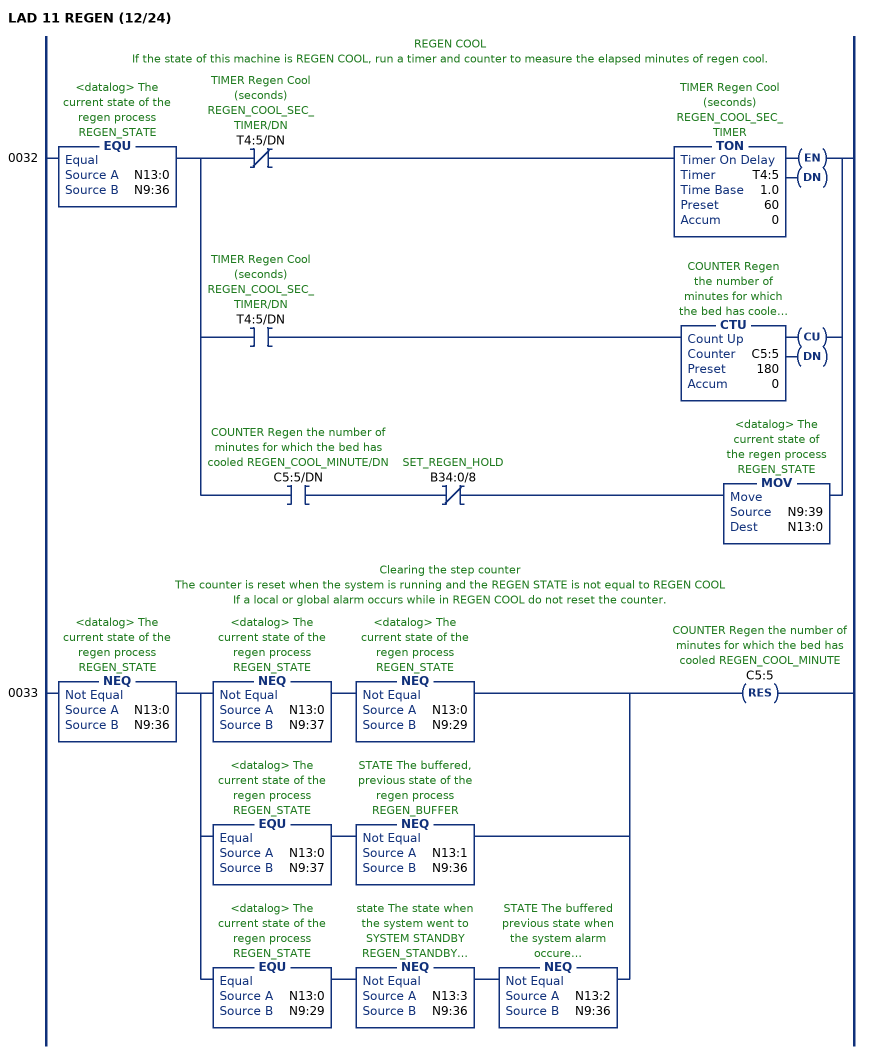
% Rung: 32 %
% REGEN COOL
% If the state of this machine is REGEN COOL, run a timer and counter to measure the elapsed minutes of regen cool. %
SOR EQU N13:0 N9:36 BST XIO T4:5/DN TON T4:5 1.0 60 0 NXB XIC T4:5/DN CTU C5:5 180 0 NXB XIC C5:5/DN XIO B34:0/8 MOV N9:39 N13:0 BND EOR
%   N13:0  REGEN_STATE  "<datalog> The current state of the regen process" %
%   N9:36  REGEN_COOL  "STATE Regen Cool" %
%   T4:5  REGEN_COOL_SEC_TIMER  "TIMER Regen Cool (seconds)" %
%   C5:5  REGEN_COOL_MINUTE  "COUNTER Regen the number of minutes for which the bed has cooled" %
%   B34:0/8  SET_REGEN_HOLD %
%   N9:39  REGEN_EQUALIZE %
% Rung: 33 %
% Clearing the step counter
% The counter is reset when the system is running and the REGEN STATE is not equal to REGEN COOL
% If a local or global alarm occurs while in REGEN COOL do not reset the counter. %
SOR NEQ N13:0 N9:36 BST NEQ N13:0 N9:37 NEQ N13:0 N9:29 NXB EQU N13:0 N9:37 NEQ N13:1 N9:36 NXB EQU N13:0 N9:29 NEQ N13:3 N9:36 NEQ N13:2 N9:36 BND RES C5:5 EOR
%   N13:0  REGEN_STATE  "<datalog> The current state of the regen process" %
%   N9:36  REGEN_COOL  "STATE Regen Cool" %
%   N9:37  REGEN_ALARM  "STATE Regen Alarm" %
%   N9:29  REGEN_IDLE %
%   N13:1  REGEN_BUFFER  "STATE The buffered, previous state of the regen process" %
%   N13:3  REGEN_STANDBY_BUFFER  "state The state when the system went to SYSTEM STANDBY" %
%   N13:2  REGEN_ALARM_BUFFER  "STATE The buffered previous state when the system alarm occured" %
%   C5:5  REGEN_COOL_MINUTE  "COUNTER Regen the number of minutes for which the bed has cooled" %

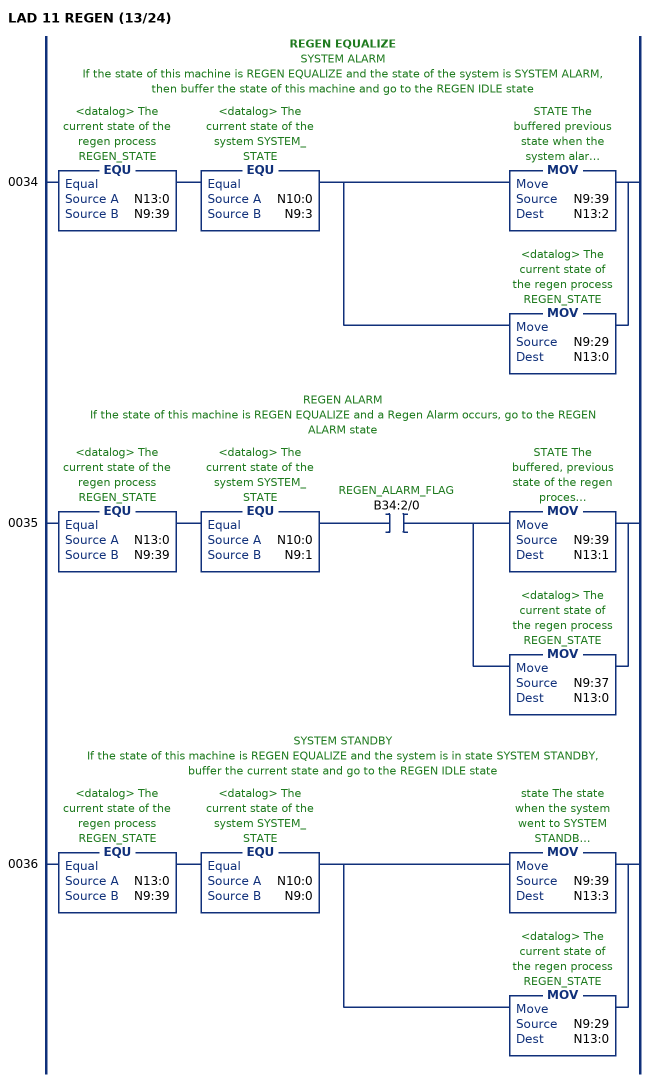
% Rung: 34 %
% TITLE: REGEN EQUALIZE %
% SYSTEM ALARM
% If the state of this machine is REGEN EQUALIZE and the state of the system is SYSTEM ALARM, then buffer the state of this machine and go to the REGEN IDLE state %
SOR EQU N13:0 N9:39 EQU N10:0 N9:3 BST MOV N9:39 N13:2 NXB MOV N9:29 N13:0 BND EOR
%   N13:0  REGEN_STATE  "<datalog> The current state of the regen process" %
%   N9:39  REGEN_EQUALIZE %
%   N10:0  SYSTEM_STATE  "<datalog> The current state of the system" %
%   N9:3  SYSTEM_ALARM  "STATE System Alarm" %
%   N13:2  REGEN_ALARM_BUFFER  "STATE The buffered previous state when the system alarm occured" %
%   N9:29  REGEN_IDLE %
% Rung: 35 %
% REGEN ALARM
% If the state of this machine is REGEN EQUALIZE and a Regen Alarm occurs, go to the REGEN ALARM state %
SOR EQU N13:0 N9:39 EQU N10:0 N9:1 XIC B34:2/0 BST MOV N9:39 N13:1 NXB MOV N9:37 N13:0 BND EOR
%   N13:0  REGEN_STATE  "<datalog> The current state of the regen process" %
%   N9:39  REGEN_EQUALIZE %
%   N10:0  SYSTEM_STATE  "<datalog> The current state of the system" %
%   N9:1  SYSTEM_PROCESS  "STATE System Process" %
%   B34:2/0  REGEN_ALARM_FLAG %
%   N13:1  REGEN_BUFFER  "STATE The buffered, previous state of the regen process" %
%   N9:37  REGEN_ALARM  "STATE Regen Alarm" %
% Rung: 36 %
% SYSTEM STANDBY
% If the state of this machine is REGEN EQUALIZE and the system is in state SYSTEM STANDBY, buffer the current state and go to the REGEN IDLE state %
SOR EQU N13:0 N9:39 EQU N10:0 N9:0 BST MOV N9:39 N13:3 NXB MOV N9:29 N13:0 BND EOR
%   N13:0  REGEN_STATE  "<datalog> The current state of the regen process" %
%   N9:39  REGEN_EQUALIZE %
%   N10:0  SYSTEM_STATE  "<datalog> The current state of the system" %
%   N9:0  SYSTEM_STANDBY  "STATE System Standby" %
%   N13:3  REGEN_STANDBY_BUFFER  "state The state when the system went to SYSTEM STANDBY" %
%   N9:29  REGEN_IDLE %

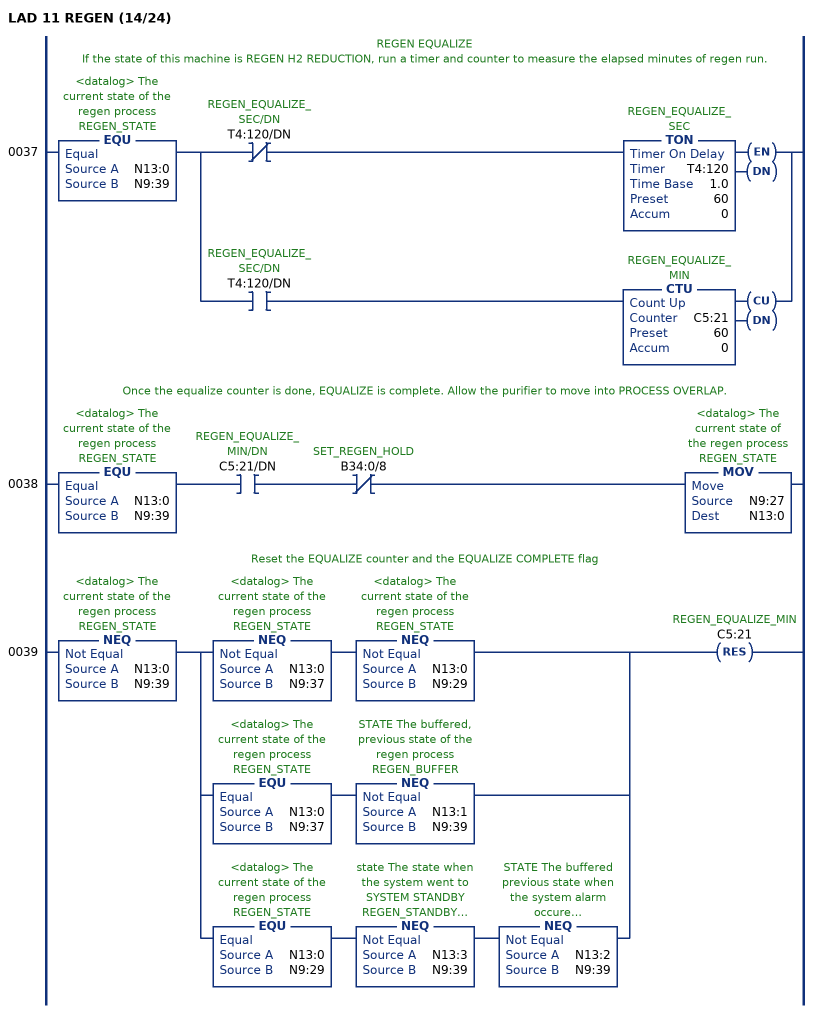
% Rung: 37 %
% REGEN EQUALIZE
% If the state of this machine is REGEN H2 REDUCTION, run a timer and counter to measure the elapsed minutes of regen run. %
SOR EQU N13:0 N9:39 BST XIO T4:120/DN TON T4:120 1.0 60 0 NXB XIC T4:120/DN CTU C5:21 60 0 BND EOR
%   N13:0  REGEN_STATE  "<datalog> The current state of the regen process" %
%   N9:39  REGEN_EQUALIZE %
%   T4:120  REGEN_EQUALIZE_SEC %
%   C5:21  REGEN_EQUALIZE_MIN %
% Rung: 38 %
% Once the equalize counter is done, EQUALIZE is complete. Allow the purifier to move into PROCESS OVERLAP. %
SOR EQU N13:0 N9:39 XIC C5:21/DN XIO B34:0/8 MOV N9:27 N13:0 EOR
%   N13:0  REGEN_STATE  "<datalog> The current state of the regen process" %
%   N9:39  REGEN_EQUALIZE %
%   C5:21  REGEN_EQUALIZE_MIN %
%   B34:0/8  SET_REGEN_HOLD %
%   N9:27  REGEN_CONDITION  "STATE Regen Idle" %
% Rung: 39 %
% Reset the EQUALIZE counter and the EQUALIZE COMPLETE flag %
SOR NEQ N13:0 N9:39 BST NEQ N13:0 N9:37 NEQ N13:0 N9:29 NXB EQU N13:0 N9:37 NEQ N13:1 N9:39 NXB EQU N13:0 N9:29 NEQ N13:3 N9:39 NEQ N13:2 N9:39 BND RES C5:21 EOR
%   N13:0  REGEN_STATE  "<datalog> The current state of the regen process" %
%   N9:39  REGEN_EQUALIZE %
%   N9:37  REGEN_ALARM  "STATE Regen Alarm" %
%   N9:29  REGEN_IDLE %
%   N13:1  REGEN_BUFFER  "STATE The buffered, previous state of the regen process" %
%   N13:3  REGEN_STANDBY_BUFFER  "state The state when the system went to SYSTEM STANDBY" %
%   N13:2  REGEN_ALARM_BUFFER  "STATE The buffered previous state when the system alarm occured" %
%   C5:21  REGEN_EQUALIZE_MIN %

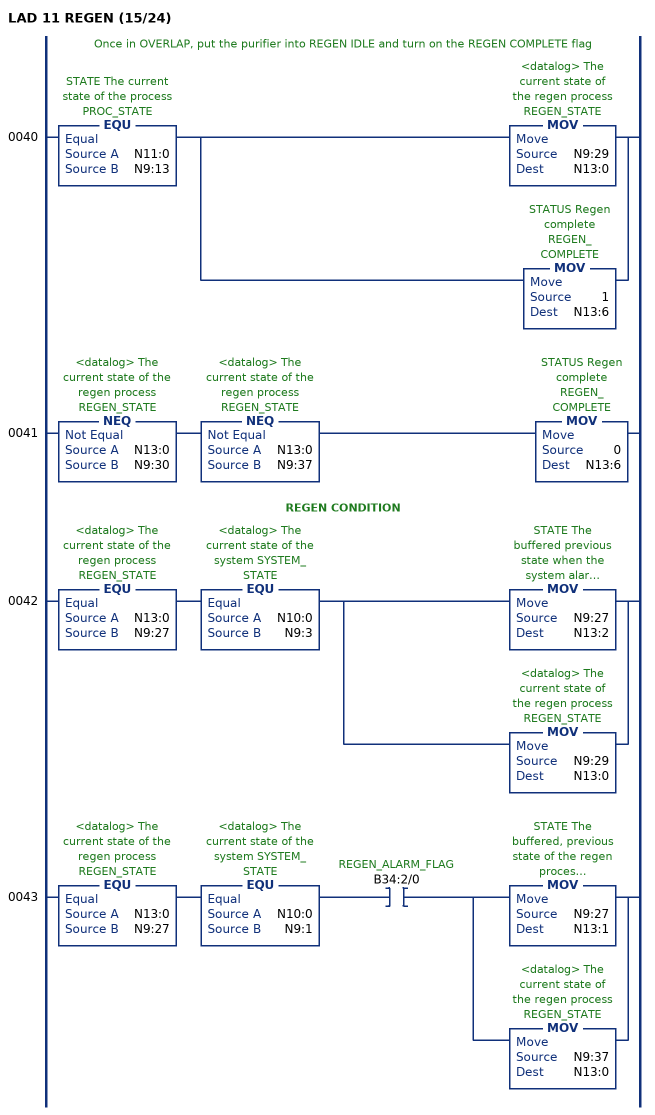
% Rung: 40 %
% Once in OVERLAP, put the purifier into REGEN IDLE and turn on the REGEN COMPLETE flag %
SOR EQU N11:0 N9:13 BST MOV N9:29 N13:0 NXB MOV 1 N13:6 BND EOR
%   N11:0  PROC_STATE  "STATE The current state of the process" %
%   N9:13  PROC_OVERLAP  "STATE Process Purify Overlap" %
%   N9:29  REGEN_IDLE %
%   N13:0  REGEN_STATE  "<datalog> The current state of the regen process" %
%   N13:6  REGEN_COMPLETE  "STATUS Regen complete" %
% Rung: 41 %
SOR NEQ N13:0 N9:30 NEQ N13:0 N9:37 MOV 0 N13:6 EOR
%   N13:0  REGEN_STATE  "<datalog> The current state of the regen process" %
%   N9:30  REGEN_STANDBY  "STATE Regen Standby" %
%   N9:37  REGEN_ALARM  "STATE Regen Alarm" %
%   N13:6  REGEN_COMPLETE  "STATUS Regen complete" %
% Rung: 42 %
% TITLE: REGEN CONDITION %
SOR EQU N13:0 N9:27 EQU N10:0 N9:3 BST MOV N9:27 N13:2 NXB MOV N9:29 N13:0 BND EOR
%   N13:0  REGEN_STATE  "<datalog> The current state of the regen process" %
%   N9:27  REGEN_CONDITION  "STATE Regen Idle" %
%   N10:0  SYSTEM_STATE  "<datalog> The current state of the system" %
%   N9:3  SYSTEM_ALARM  "STATE System Alarm" %
%   N13:2  REGEN_ALARM_BUFFER  "STATE The buffered previous state when the system alarm occured" %
%   N9:29  REGEN_IDLE %
% Rung: 43 %
SOR EQU N13:0 N9:27 EQU N10:0 N9:1 XIC B34:2/0 BST MOV N9:27 N13:1 NXB MOV N9:37 N13:0 BND EOR
%   N13:0  REGEN_STATE  "<datalog> The current state of the regen process" %
%   N9:27  REGEN_CONDITION  "STATE Regen Idle" %
%   N10:0  SYSTEM_STATE  "<datalog> The current state of the system" %
%   N9:1  SYSTEM_PROCESS  "STATE System Process" %
%   B34:2/0  REGEN_ALARM_FLAG %
%   N13:1  REGEN_BUFFER  "STATE The buffered, previous state of the regen process" %
%   N9:37  REGEN_ALARM  "STATE Regen Alarm" %

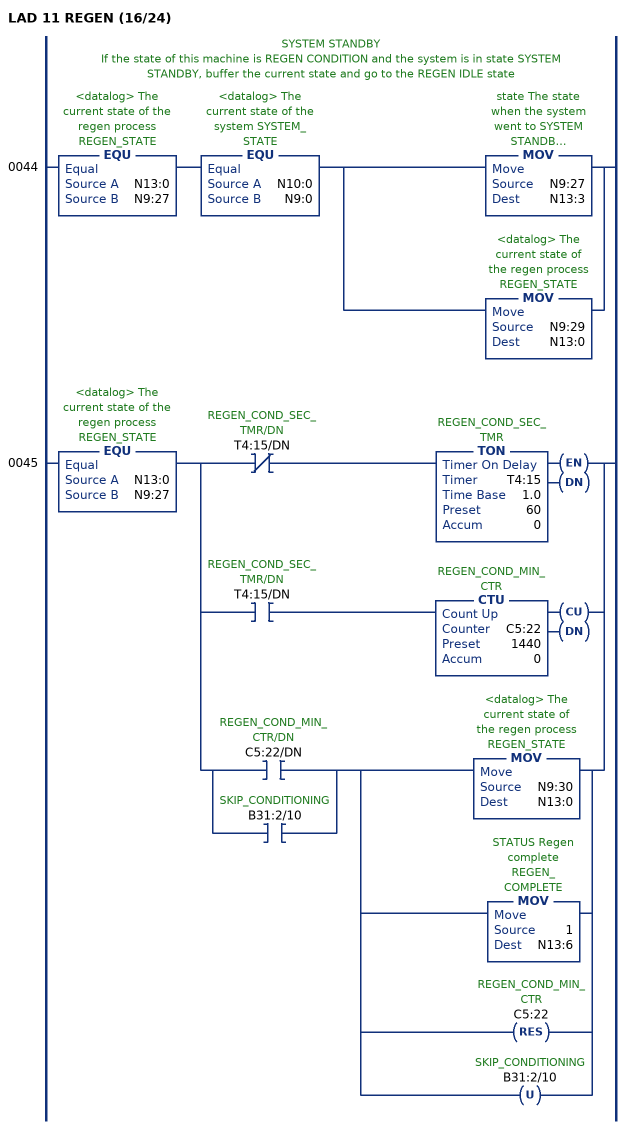
% Rung: 44 %
% SYSTEM STANDBY
% If the state of this machine is REGEN CONDITION and the system is in state SYSTEM STANDBY, buffer the current state and go to the REGEN IDLE state %
SOR EQU N13:0 N9:27 EQU N10:0 N9:0 BST MOV N9:27 N13:3 NXB MOV N9:29 N13:0 BND EOR
%   N13:0  REGEN_STATE  "<datalog> The current state of the regen process" %
%   N9:27  REGEN_CONDITION  "STATE Regen Idle" %
%   N10:0  SYSTEM_STATE  "<datalog> The current state of the system" %
%   N9:0  SYSTEM_STANDBY  "STATE System Standby" %
%   N13:3  REGEN_STANDBY_BUFFER  "state The state when the system went to SYSTEM STANDBY" %
%   N9:29  REGEN_IDLE %
% Rung: 45 %
SOR EQU N13:0 N9:27 BST XIO T4:15/DN TON T4:15 1.0 60 0 NXB XIC T4:15/DN CTU C5:22 1440 0 NXB BST XIC C5:22/DN NXB XIC B31:2/10 BND BST MOV N9:30 N13:0 NXB MOV 1 N13:6 NXB RES C5:22 NXB OTU B31:2/10 BND BND EOR
%   N13:0  REGEN_STATE  "<datalog> The current state of the regen process" %
%   N9:27  REGEN_CONDITION  "STATE Regen Idle" %
%   T4:15  REGEN_COND_SEC_TMR %
%   C5:22  REGEN_COND_MIN_CTR %
%   B31:2/10  SKIP_CONDITIONING %
%   N9:30  REGEN_STANDBY  "STATE Regen Standby" %
%   N13:6  REGEN_COMPLETE  "STATUS Regen complete" %

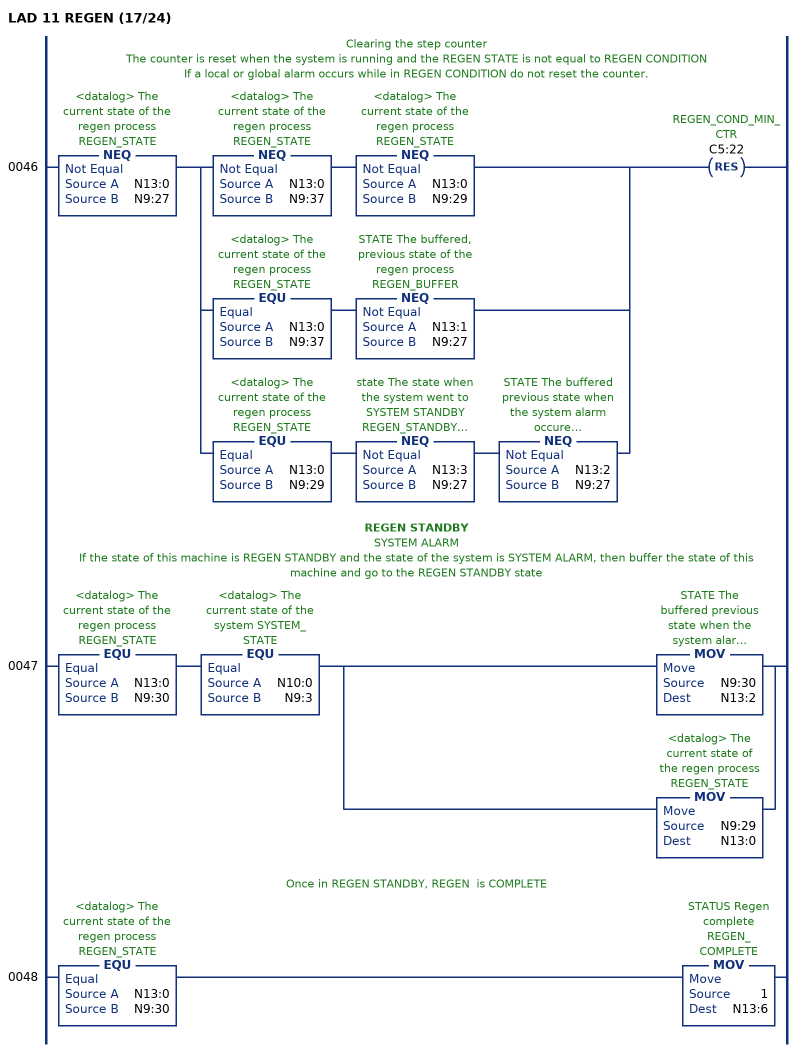
% Rung: 46 %
% Clearing the step counter
% The counter is reset when the system is running and the REGEN STATE is not equal to REGEN CONDITION
% If a local or global alarm occurs while in REGEN CONDITION do not reset the counter. %
SOR NEQ N13:0 N9:27 BST NEQ N13:0 N9:37 NEQ N13:0 N9:29 NXB EQU N13:0 N9:37 NEQ N13:1 N9:27 NXB EQU N13:0 N9:29 NEQ N13:3 N9:27 NEQ N13:2 N9:27 BND RES C5:22 EOR
%   N13:0  REGEN_STATE  "<datalog> The current state of the regen process" %
%   N9:27  REGEN_CONDITION  "STATE Regen Idle" %
%   N9:37  REGEN_ALARM  "STATE Regen Alarm" %
%   N9:29  REGEN_IDLE %
%   N13:1  REGEN_BUFFER  "STATE The buffered, previous state of the regen process" %
%   N13:3  REGEN_STANDBY_BUFFER  "state The state when the system went to SYSTEM STANDBY" %
%   N13:2  REGEN_ALARM_BUFFER  "STATE The buffered previous state when the system alarm occured" %
%   C5:22  REGEN_COND_MIN_CTR %
% Rung: 47 %
% TITLE: REGEN STANDBY %
% SYSTEM ALARM
% If the state of this machine is REGEN STANDBY and the state of the system is SYSTEM ALARM, then buffer the state of this machine and go to the REGEN STANDBY state %
SOR EQU N13:0 N9:30 EQU N10:0 N9:3 BST MOV N9:30 N13:2 NXB MOV N9:29 N13:0 BND EOR
%   N13:0  REGEN_STATE  "<datalog> The current state of the regen process" %
%   N9:30  REGEN_STANDBY  "STATE Regen Standby" %
%   N10:0  SYSTEM_STATE  "<datalog> The current state of the system" %
%   N9:3  SYSTEM_ALARM  "STATE System Alarm" %
%   N13:2  REGEN_ALARM_BUFFER  "STATE The buffered previous state when the system alarm occured" %
%   N9:29  REGEN_IDLE %
% Rung: 48 %
% Once in REGEN STANDBY, REGEN  is COMPLETE %
SOR EQU N13:0 N9:30 MOV 1 N13:6 EOR
%   N13:0  REGEN_STATE  "<datalog> The current state of the regen process" %
%   N9:30  REGEN_STANDBY  "STATE Regen Standby" %
%   N13:6  REGEN_COMPLETE  "STATUS Regen complete" %

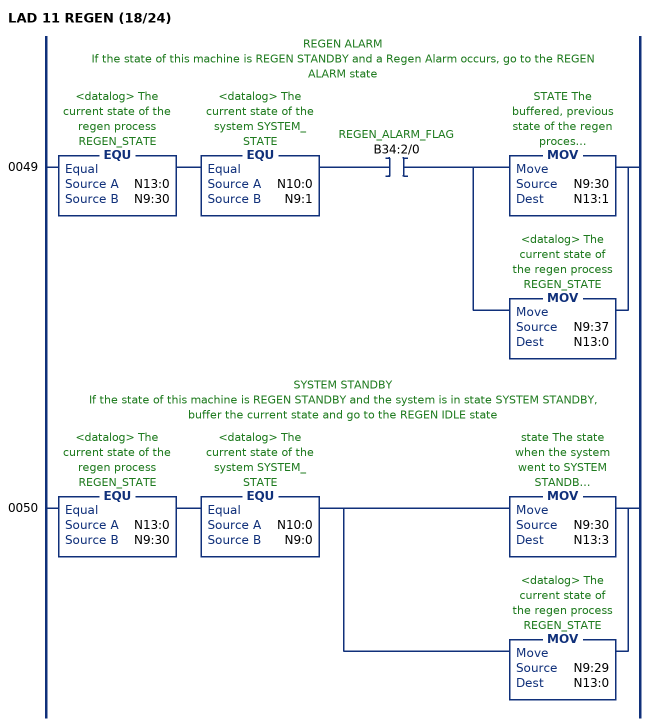
% Rung: 49 %
% REGEN ALARM
% If the state of this machine is REGEN STANDBY and a Regen Alarm occurs, go to the REGEN ALARM state %
SOR EQU N13:0 N9:30 EQU N10:0 N9:1 XIC B34:2/0 BST MOV N9:30 N13:1 NXB MOV N9:37 N13:0 BND EOR
%   N13:0  REGEN_STATE  "<datalog> The current state of the regen process" %
%   N9:30  REGEN_STANDBY  "STATE Regen Standby" %
%   N10:0  SYSTEM_STATE  "<datalog> The current state of the system" %
%   N9:1  SYSTEM_PROCESS  "STATE System Process" %
%   B34:2/0  REGEN_ALARM_FLAG %
%   N13:1  REGEN_BUFFER  "STATE The buffered, previous state of the regen process" %
%   N9:37  REGEN_ALARM  "STATE Regen Alarm" %
% Rung: 50 %
% SYSTEM STANDBY
% If the state of this machine is REGEN STANDBY and the system is in state SYSTEM STANDBY, buffer the current state and go to the REGEN IDLE state %
SOR EQU N13:0 N9:30 EQU N10:0 N9:0 BST MOV N9:30 N13:3 NXB MOV N9:29 N13:0 BND EOR
%   N13:0  REGEN_STATE  "<datalog> The current state of the regen process" %
%   N9:30  REGEN_STANDBY  "STATE Regen Standby" %
%   N10:0  SYSTEM_STATE  "<datalog> The current state of the system" %
%   N9:0  SYSTEM_STANDBY  "STATE System Standby" %
%   N13:3  REGEN_STANDBY_BUFFER  "state The state when the system went to SYSTEM STANDBY" %
%   N9:29  REGEN_IDLE %

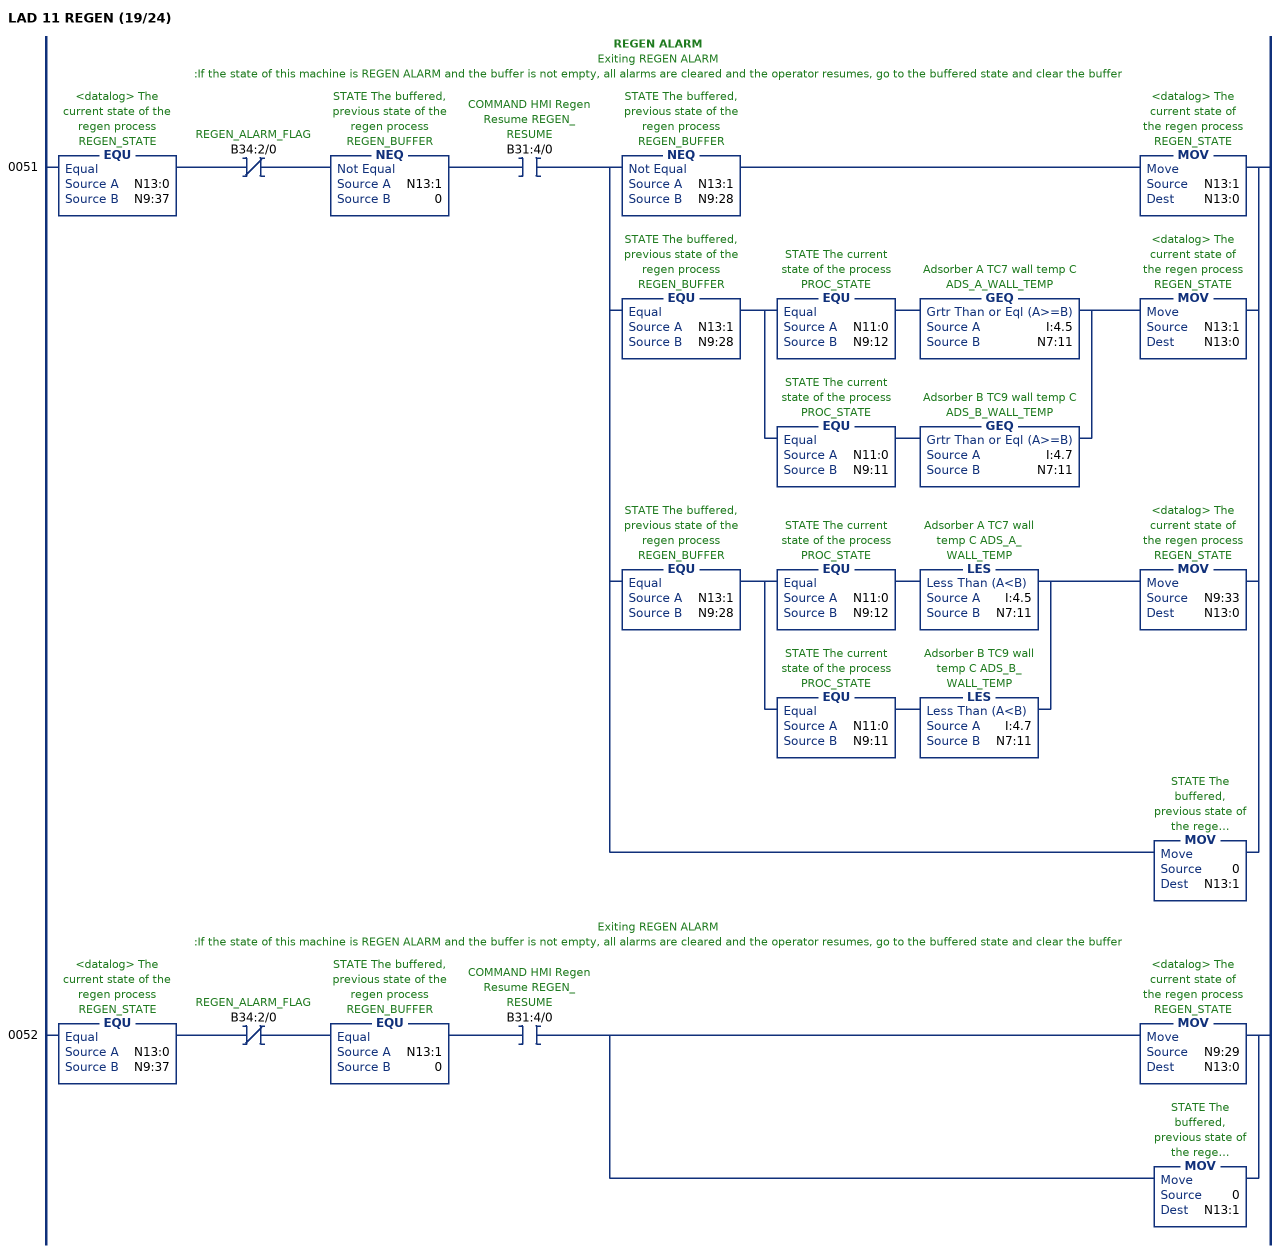
% Rung: 51 %
% TITLE: REGEN ALARM %
% Exiting REGEN ALARM
% :If the state of this machine is REGEN ALARM and the buffer is not empty, all alarms are cleared and the operator resumes, go to the buffered state and clear the buffer %
SOR EQU N13:0 N9:37 XIO B34:2/0 NEQ N13:1 0 XIC B31:4/0 BST NEQ N13:1 N9:28 MOV N13:1 N13:0 NXB EQU N13:1 N9:28 BST EQU N11:0 N9:12 GEQ I:4.5 N7:11 NXB EQU N11:0 N9:11 GEQ I:4.7 N7:11 BND MOV N13:1 N13:0 NXB EQU N13:1 N9:28 BST EQU N11:0 N9:12 LES I:4.5 N7:11 NXB EQU N11:0 N9:11 LES I:4.7 N7:11 BND MOV N9:33 N13:0 NXB MOV 0 N13:1 BND EOR
%   N13:0  REGEN_STATE  "<datalog> The current state of the regen process" %
%   N9:37  REGEN_ALARM  "STATE Regen Alarm" %
%   B34:2/0  REGEN_ALARM_FLAG %
%   N13:1  REGEN_BUFFER  "STATE The buffered, previous state of the regen process" %
%   B31:4/0  REGEN_RESUME  "COMMAND HMI Regen Resume" %
%   N9:28  REGEN_RUN %
%   N11:0  PROC_STATE  "STATE The current state of the process" %
%   N9:12  PROC_REGEN_A  "STATE Process Purify B" %
%   I:4.5  ADS_A_WALL_TEMP  "Adsorber A TC7 wall temp C" %
%   N7:11  ADS_BED_TEMP_HIGH  "CONFIG The temp at which the regen process may continue" %
%   N9:11  PROC_REGEN_B  "STATE Process Purify A" %
%   I:4.7  ADS_B_WALL_TEMP  "Adsorber B TC9 wall temp C" %
%   N9:33  REGEN_HEAT_BED  "STATE Regen Heat wall" %
% Rung: 52 %
% Exiting REGEN ALARM
% :If the state of this machine is REGEN ALARM and the buffer is not empty, all alarms are cleared and the operator resumes, go to the buffered state and clear the buffer %
SOR EQU N13:0 N9:37 XIO B34:2/0 EQU N13:1 0 XIC B31:4/0 BST MOV N9:29 N13:0 NXB MOV 0 N13:1 BND EOR
%   N13:0  REGEN_STATE  "<datalog> The current state of the regen process" %
%   N9:37  REGEN_ALARM  "STATE Regen Alarm" %
%   B34:2/0  REGEN_ALARM_FLAG %
%   N13:1  REGEN_BUFFER  "STATE The buffered, previous state of the regen process" %
%   B31:4/0  REGEN_RESUME  "COMMAND HMI Regen Resume" %
%   N9:29  REGEN_IDLE %

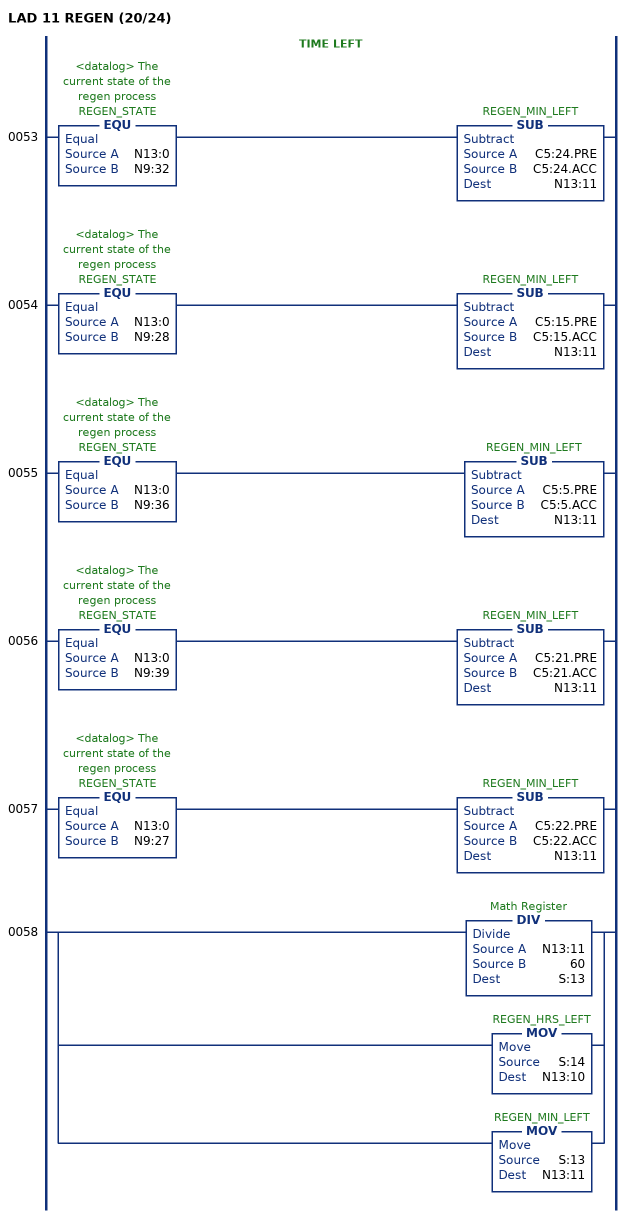
% Rung: 53 %
% TITLE: TIME LEFT %
SOR EQU N13:0 N9:32 SUB C5:24.PRE C5:24.ACC N13:11 EOR
%   N13:0  REGEN_STATE  "<datalog> The current state of the regen process" %
%   N9:32  REGEN_VENT  "STATE Regen Vent" %
%   C5:24  REGEN_VENT_MIN_CTR %
%   N13:11  REGEN_MIN_LEFT %
% Rung: 54 %
SOR EQU N13:0 N9:28 SUB C5:15.PRE C5:15.ACC N13:11 EOR
%   N13:0  REGEN_STATE  "<datalog> The current state of the regen process" %
%   N9:28  REGEN_RUN %
%   C5:15  REGEN_RUN_MINUTE %
%   N13:11  REGEN_MIN_LEFT %
% Rung: 55 %
SOR EQU N13:0 N9:36 SUB C5:5.PRE C5:5.ACC N13:11 EOR
%   N13:0  REGEN_STATE  "<datalog> The current state of the regen process" %
%   N9:36  REGEN_COOL  "STATE Regen Cool" %
%   C5:5  REGEN_COOL_MINUTE  "COUNTER Regen the number of minutes for which the bed has cooled" %
%   N13:11  REGEN_MIN_LEFT %
% Rung: 56 %
SOR EQU N13:0 N9:39 SUB C5:21.PRE C5:21.ACC N13:11 EOR
%   N13:0  REGEN_STATE  "<datalog> The current state of the regen process" %
%   N9:39  REGEN_EQUALIZE %
%   C5:21  REGEN_EQUALIZE_MIN %
%   N13:11  REGEN_MIN_LEFT %
% Rung: 57 %
SOR EQU N13:0 N9:27 SUB C5:22.PRE C5:22.ACC N13:11 EOR
%   N13:0  REGEN_STATE  "<datalog> The current state of the regen process" %
%   N9:27  REGEN_CONDITION  "STATE Regen Idle" %
%   C5:22  REGEN_COND_MIN_CTR %
%   N13:11  REGEN_MIN_LEFT %
% Rung: 58 %
SOR BST DIV N13:11 60 S:13 NXB MOV S:14 N13:10 NXB MOV S:13 N13:11 BND EOR
%   N13:11  REGEN_MIN_LEFT %
%   S:13  "Math Register" %
%   S:14  "Math Register" %
%   N13:10  REGEN_HRS_LEFT %

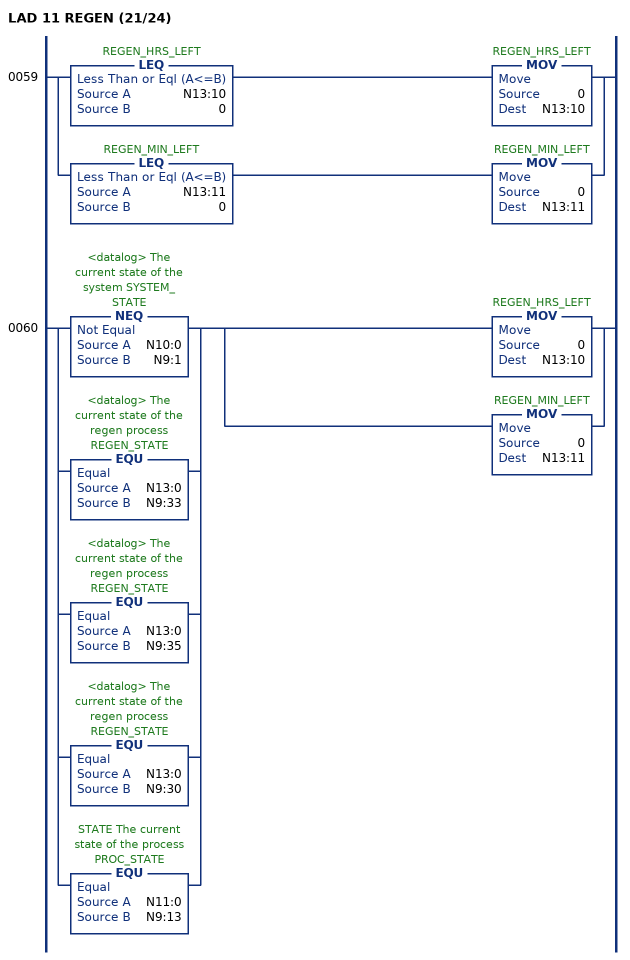
% Rung: 59 %
SOR BST LEQ N13:10 0 MOV 0 N13:10 NXB LEQ N13:11 0 MOV 0 N13:11 BND EOR
%   N13:10  REGEN_HRS_LEFT %
%   N13:11  REGEN_MIN_LEFT %
% Rung: 60 %
SOR BST NEQ N10:0 N9:1 NXB EQU N13:0 N9:33 NXB EQU N13:0 N9:35 NXB EQU N13:0 N9:30 NXB EQU N11:0 N9:13 BND BST MOV 0 N13:10 NXB MOV 0 N13:11 BND EOR
%   N10:0  SYSTEM_STATE  "<datalog> The current state of the system" %
%   N9:1  SYSTEM_PROCESS  "STATE System Process" %
%   N13:0  REGEN_STATE  "<datalog> The current state of the regen process" %
%   N9:33  REGEN_HEAT_BED  "STATE Regen Heat wall" %
%   N9:35  REGEN_COOL_WALL  "STATE Regen Cool wall" %
%   N9:30  REGEN_STANDBY  "STATE Regen Standby" %
%   N11:0  PROC_STATE  "STATE The current state of the process" %
%   N9:13  PROC_OVERLAP  "STATE Process Purify Overlap" %
%   N13:10  REGEN_HRS_LEFT %
%   N13:11  REGEN_MIN_LEFT %

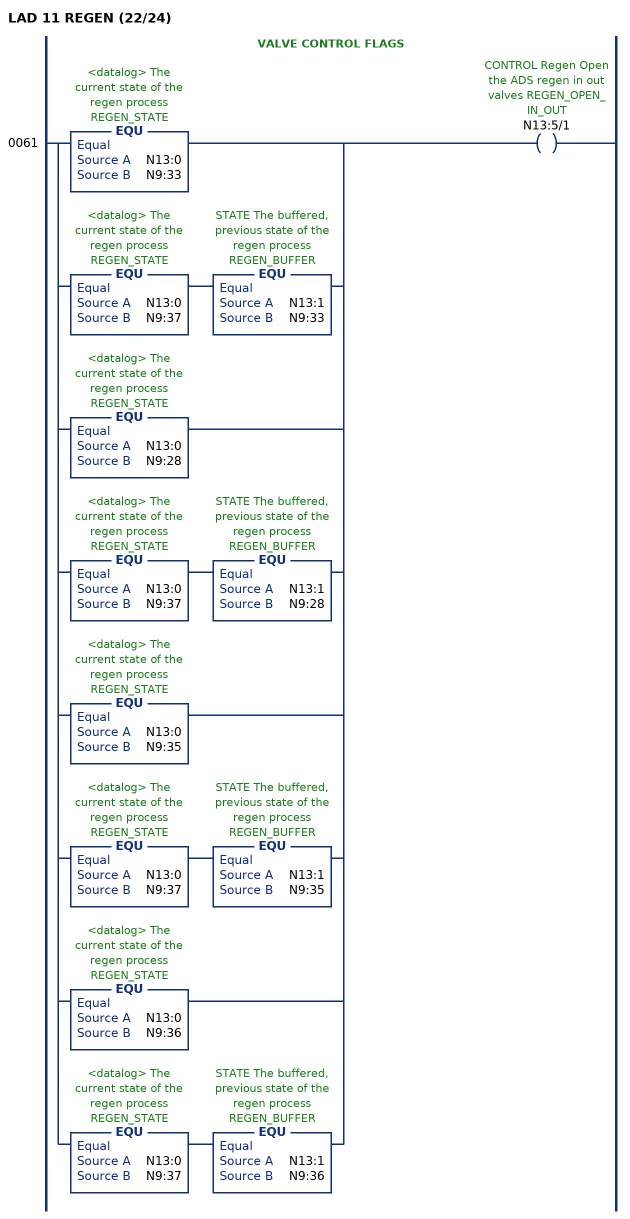
% Rung: 61 %
% TITLE: VALVE CONTROL FLAGS %
SOR BST EQU N13:0 N9:33 NXB EQU N13:0 N9:37 EQU N13:1 N9:33 NXB EQU N13:0 N9:28 NXB EQU N13:0 N9:37 EQU N13:1 N9:28 NXB EQU N13:0 N9:35 NXB EQU N13:0 N9:37 EQU N13:1 N9:35 NXB EQU N13:0 N9:36 NXB EQU N13:0 N9:37 EQU N13:1 N9:36 BND OTE N13:5/1 EOR
%   N13:0  REGEN_STATE  "<datalog> The current state of the regen process" %
%   N9:33  REGEN_HEAT_BED  "STATE Regen Heat wall" %
%   N9:37  REGEN_ALARM  "STATE Regen Alarm" %
%   N13:1  REGEN_BUFFER  "STATE The buffered, previous state of the regen process" %
%   N9:28  REGEN_RUN %
%   N9:35  REGEN_COOL_WALL  "STATE Regen Cool wall" %
%   N9:36  REGEN_COOL  "STATE Regen Cool" %
%   N13:5/1  REGEN_OPEN_IN_OUT  "CONTROL Regen Open the ADS regen in out valves" %

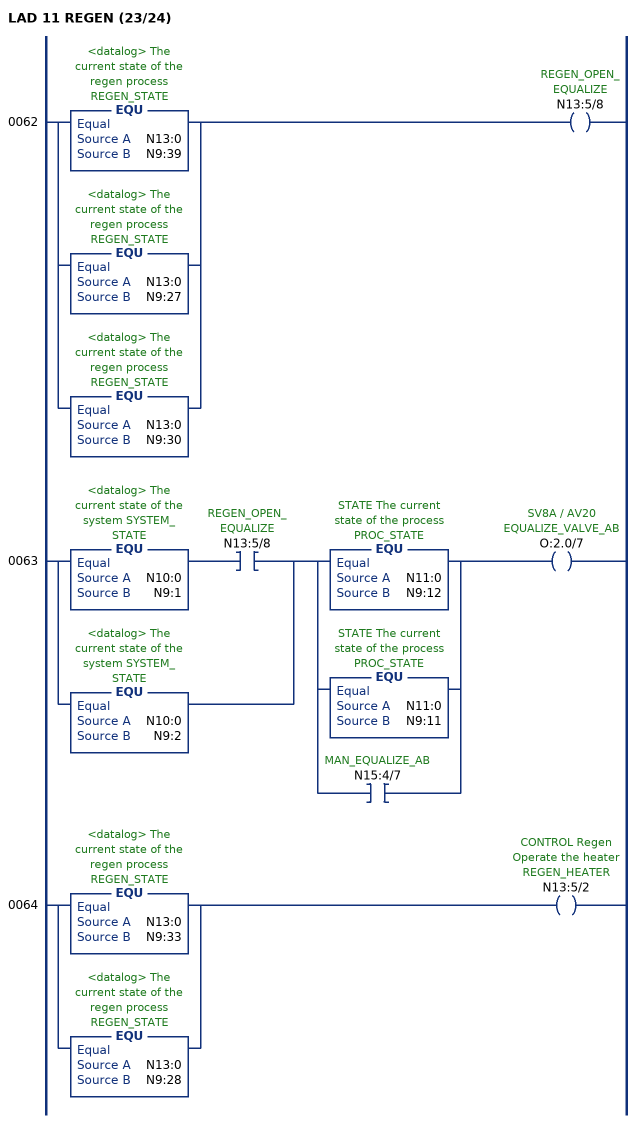
% Rung: 62 %
SOR BST EQU N13:0 N9:39 NXB EQU N13:0 N9:27 NXB EQU N13:0 N9:30 BND OTE N13:5/8 EOR
%   N13:0  REGEN_STATE  "<datalog> The current state of the regen process" %
%   N9:39  REGEN_EQUALIZE %
%   N9:27  REGEN_CONDITION  "STATE Regen Idle" %
%   N9:30  REGEN_STANDBY  "STATE Regen Standby" %
%   N13:5/8  REGEN_OPEN_EQUALIZE %
% Rung: 63 %
SOR BST EQU N10:0 N9:1 XIC N13:5/8 NXB EQU N10:0 N9:2 BND BST EQU N11:0 N9:12 NXB EQU N11:0 N9:11 NXB XIC N15:4/7 BND OTE O:2.0/7 EOR
%   N10:0  SYSTEM_STATE  "<datalog> The current state of the system" %
%   N9:1  SYSTEM_PROCESS  "STATE System Process" %
%   N13:5/8  REGEN_OPEN_EQUALIZE %
%   N9:2  SYSTEM_MANUAL  "STATE System Manual" %
%   N11:0  PROC_STATE  "STATE The current state of the process" %
%   N9:12  PROC_REGEN_A  "STATE Process Purify B" %
%   N9:11  PROC_REGEN_B  "STATE Process Purify A" %
%   N15:4/7  MAN_EQUALIZE_AB %
%   O:2.0/7  EQUALIZE_VALVE_AB  "SV8A / AV20" %
% Rung: 64 %
SOR BST EQU N13:0 N9:33 NXB EQU N13:0 N9:28 BND OTE N13:5/2 EOR
%   N13:0  REGEN_STATE  "<datalog> The current state of the regen process" %
%   N9:33  REGEN_HEAT_BED  "STATE Regen Heat wall" %
%   N9:28  REGEN_RUN %
%   N13:5/2  REGEN_HEATER  "CONTROL Regen Operate the heater" %

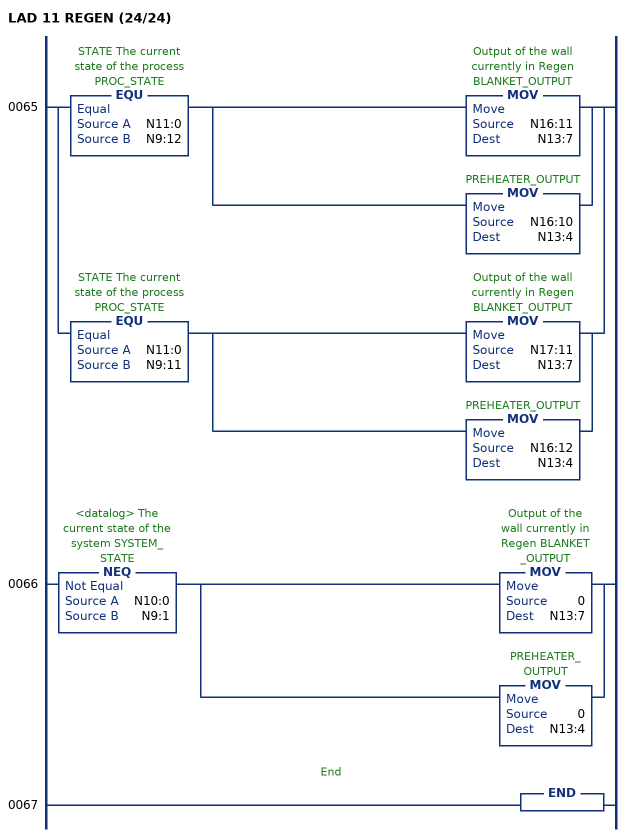
% Rung: 65 %
SOR BST EQU N11:0 N9:12 BST MOV N16:11 N13:7 NXB MOV N16:10 N13:4 BND NXB EQU N11:0 N9:11 BST MOV N17:11 N13:7 NXB MOV N16:12 N13:4 BND BND EOR
%   N11:0  PROC_STATE  "STATE The current state of the process" %
%   N9:12  PROC_REGEN_A  "STATE Process Purify B" %
%   N16:11  ADS_A_BLNKT_OUTPUT  "CONTROL ADS A Blanket output (percent)" %
%   N13:7  BLANKET_OUTPUT  "Output of the wall currently in Regen" %
%   N16:10  ADS_A_PH_OUTPUT  "<datalog> Adsorber A heater duty cycle %" %
%   N13:4  PREHEATER_OUTPUT %
%   N9:11  PROC_REGEN_B  "STATE Process Purify A" %
%   N17:11  ADS_B_BLNKT_OUTPUT  "CONTROL ADS A Blanket output" %
%   N16:12  ADS_B_PH_OUTPUT  "<datalog> Adsorber B heater duty cycle %" %
% Rung: 66 %
SOR NEQ N10:0 N9:1 BST MOV 0 N13:7 NXB MOV 0 N13:4 BND EOR
%   N10:0  SYSTEM_STATE  "<datalog> The current state of the system" %
%   N9:1  SYSTEM_PROCESS  "STATE System Process" %
%   N13:7  BLANKET_OUTPUT  "Output of the wall currently in Regen" %
%   N13:4  PREHEATER_OUTPUT %
% Rung: 67 %
% End %
SOR END EOR

LADDER 12 "REGEN_FLT"    % regen alarms and warnings %
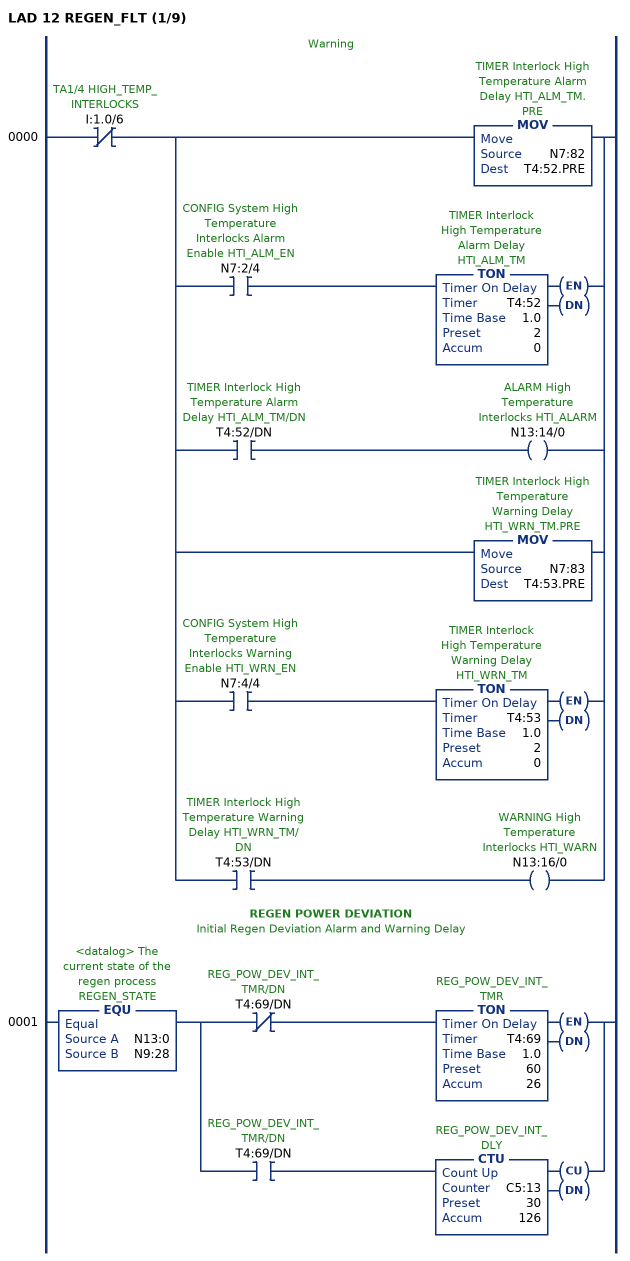
% Rung: 0 %
% Warning %
SOR XIO I:1.0/6 BST MOV N7:82 T4:52.PRE NXB XIC N7:2/4 TON T4:52 1.0 2 0 NXB XIC T4:52/DN OTE N13:14/0 NXB MOV N7:83 T4:53.PRE NXB XIC N7:4/4 TON T4:53 1.0 2 0 NXB XIC T4:53/DN OTE N13:16/0 BND EOR
%   I:1.0/6  HIGH_TEMP_INTERLOCKS  "TA1/4" %
%   N7:82  HTI_ALM_DY  "CONFIG Interlocks High Temp Alarm Delay" %
%   T4:52  HTI_ALM_TM  "TIMER Interlock High Temperature Alarm Delay" %
%   N7:2/4  HTI_ALM_EN  "CONFIG System High Temperature Interlocks Alarm Enable" %
%   N13:14/0  HTI_ALARM  "ALARM High Temperature Interlocks" %
%   N7:83  HTI_WRN_DY  "CONFIG Interlocks High Temp Warning Delay" %
%   T4:53  HTI_WRN_TM  "TIMER Interlock High Temperature Warning Delay" %
%   N7:4/4  HTI_WRN_EN  "CONFIG System High Temperature Interlocks Warning Enable" %
%   N13:16/0  HTI_WARN  "WARNING High Temperature Interlocks" %
% Rung: 1 %
% TITLE: REGEN POWER DEVIATION %
% Initial Regen Deviation Alarm and Warning Delay %
SOR EQU N13:0 N9:28 BST XIO T4:69/DN TON T4:69 1.0 60 26 NXB XIC T4:69/DN CTU C5:13 30 126 BND EOR
%   N13:0  REGEN_STATE  "<datalog> The current state of the regen process" %
%   N9:28  REGEN_RUN %
%   T4:69  REG_POW_DEV_INT_TMR %
%   C5:13  REG_POW_DEV_INT_DLY %

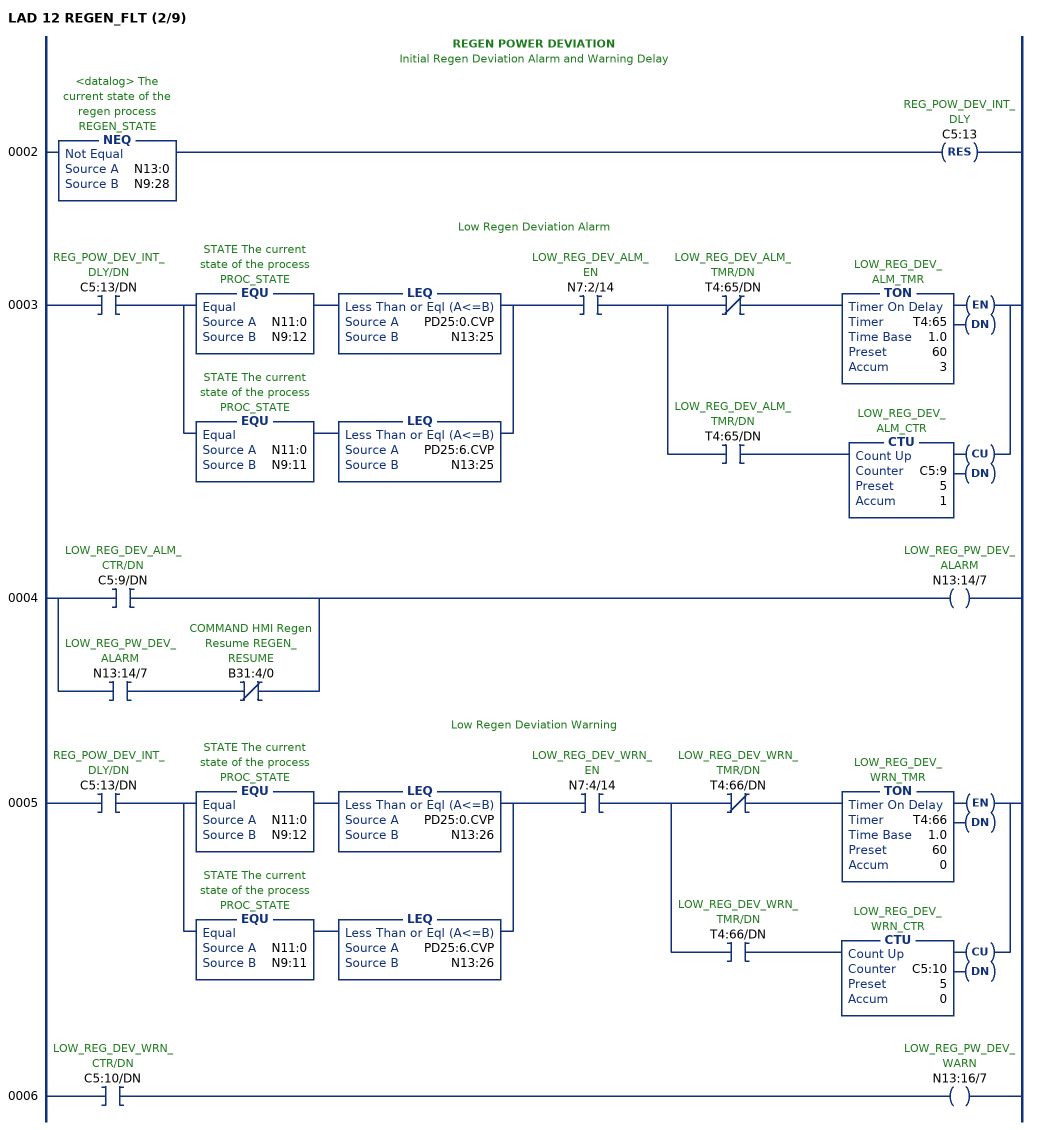
% Rung: 2 %
% TITLE: REGEN POWER DEVIATION %
% Initial Regen Deviation Alarm and Warning Delay %
SOR NEQ N13:0 N9:28 RES C5:13 EOR
%   N13:0  REGEN_STATE  "<datalog> The current state of the regen process" %
%   N9:28  REGEN_RUN %
%   C5:13  REG_POW_DEV_INT_DLY %
% Rung: 3 %
% Low Regen Deviation Alarm %
SOR XIC C5:13/DN BST EQU N11:0 N9:12 LEQ PD25:0.CVP N13:25 NXB EQU N11:0 N9:11 LEQ PD25:6.CVP N13:25 BND XIC N7:2/14 BST XIO T4:65/DN TON T4:65 1.0 60 3 NXB XIC T4:65/DN CTU C5:9 5 1 BND EOR
%   C5:13  REG_POW_DEV_INT_DLY %
%   N11:0  PROC_STATE  "STATE The current state of the process" %
%   N9:12  PROC_REGEN_A  "STATE Process Purify B" %
%   N13:25  LOW_REG_DEV_ALM_SP %
%   N9:11  PROC_REGEN_B  "STATE Process Purify A" %
%   N7:2/14  LOW_REG_DEV_ALM_EN %
%   T4:65  LOW_REG_DEV_ALM_TMR %
%   C5:9  LOW_REG_DEV_ALM_CTR %
% Rung: 4 %
SOR BST XIC C5:9/DN NXB XIC N13:14/7 XIO B31:4/0 BND OTE N13:14/7 EOR
%   C5:9  LOW_REG_DEV_ALM_CTR %
%   N13:14/7  LOW_REG_PW_DEV_ALARM %
%   B31:4/0  REGEN_RESUME  "COMMAND HMI Regen Resume" %
% Rung: 5 %
% Low Regen Deviation Warning %
SOR XIC C5:13/DN BST EQU N11:0 N9:12 LEQ PD25:0.CVP N13:26 NXB EQU N11:0 N9:11 LEQ PD25:6.CVP N13:26 BND XIC N7:4/14 BST XIO T4:66/DN TON T4:66 1.0 60 0 NXB XIC T4:66/DN CTU C5:10 5 0 BND EOR
%   C5:13  REG_POW_DEV_INT_DLY %
%   N11:0  PROC_STATE  "STATE The current state of the process" %
%   N9:12  PROC_REGEN_A  "STATE Process Purify B" %
%   N13:26  LOW_REG_DEV_WRN_SP %
%   N9:11  PROC_REGEN_B  "STATE Process Purify A" %
%   N7:4/14  LOW_REG_DEV_WRN_EN %
%   T4:66  LOW_REG_DEV_WRN_TMR %
%   C5:10  LOW_REG_DEV_WRN_CTR %
% Rung: 6 %
SOR XIC C5:10/DN OTE N13:16/7 EOR
%   C5:10  LOW_REG_DEV_WRN_CTR %
%   N13:16/7  LOW_REG_PW_DEV_WARN %

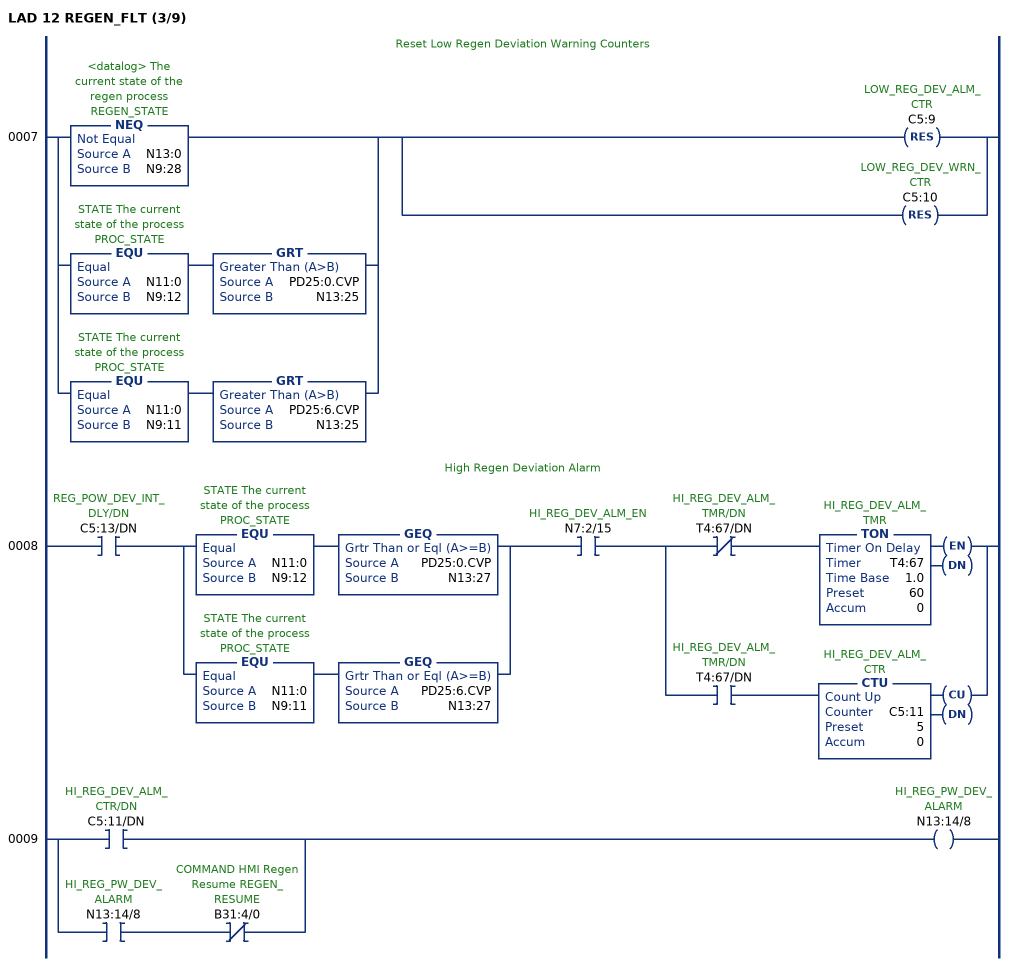
% Rung: 7 %
% Reset Low Regen Deviation Warning Counters %
SOR BST NEQ N13:0 N9:28 NXB EQU N11:0 N9:12 GRT PD25:0.CVP N13:25 NXB EQU N11:0 N9:11 GRT PD25:6.CVP N13:25 BND BST RES C5:9 NXB RES C5:10 BND EOR
%   N13:0  REGEN_STATE  "<datalog> The current state of the regen process" %
%   N9:28  REGEN_RUN %
%   N11:0  PROC_STATE  "STATE The current state of the process" %
%   N9:12  PROC_REGEN_A  "STATE Process Purify B" %
%   N13:25  LOW_REG_DEV_ALM_SP %
%   N9:11  PROC_REGEN_B  "STATE Process Purify A" %
%   C5:9  LOW_REG_DEV_ALM_CTR %
%   C5:10  LOW_REG_DEV_WRN_CTR %
% Rung: 8 %
% High Regen Deviation Alarm %
SOR XIC C5:13/DN BST EQU N11:0 N9:12 GEQ PD25:0.CVP N13:27 NXB EQU N11:0 N9:11 GEQ PD25:6.CVP N13:27 BND XIC N7:2/15 BST XIO T4:67/DN TON T4:67 1.0 60 0 NXB XIC T4:67/DN CTU C5:11 5 0 BND EOR
%   C5:13  REG_POW_DEV_INT_DLY %
%   N11:0  PROC_STATE  "STATE The current state of the process" %
%   N9:12  PROC_REGEN_A  "STATE Process Purify B" %
%   N13:27  HI_REG_DEV_ALM_SP %
%   N9:11  PROC_REGEN_B  "STATE Process Purify A" %
%   N7:2/15  HI_REG_DEV_ALM_EN %
%   T4:67  HI_REG_DEV_ALM_TMR %
%   C5:11  HI_REG_DEV_ALM_CTR %
% Rung: 9 %
SOR BST XIC C5:11/DN NXB XIC N13:14/8 XIO B31:4/0 BND OTE N13:14/8 EOR
%   C5:11  HI_REG_DEV_ALM_CTR %
%   N13:14/8  HI_REG_PW_DEV_ALARM %
%   B31:4/0  REGEN_RESUME  "COMMAND HMI Regen Resume" %

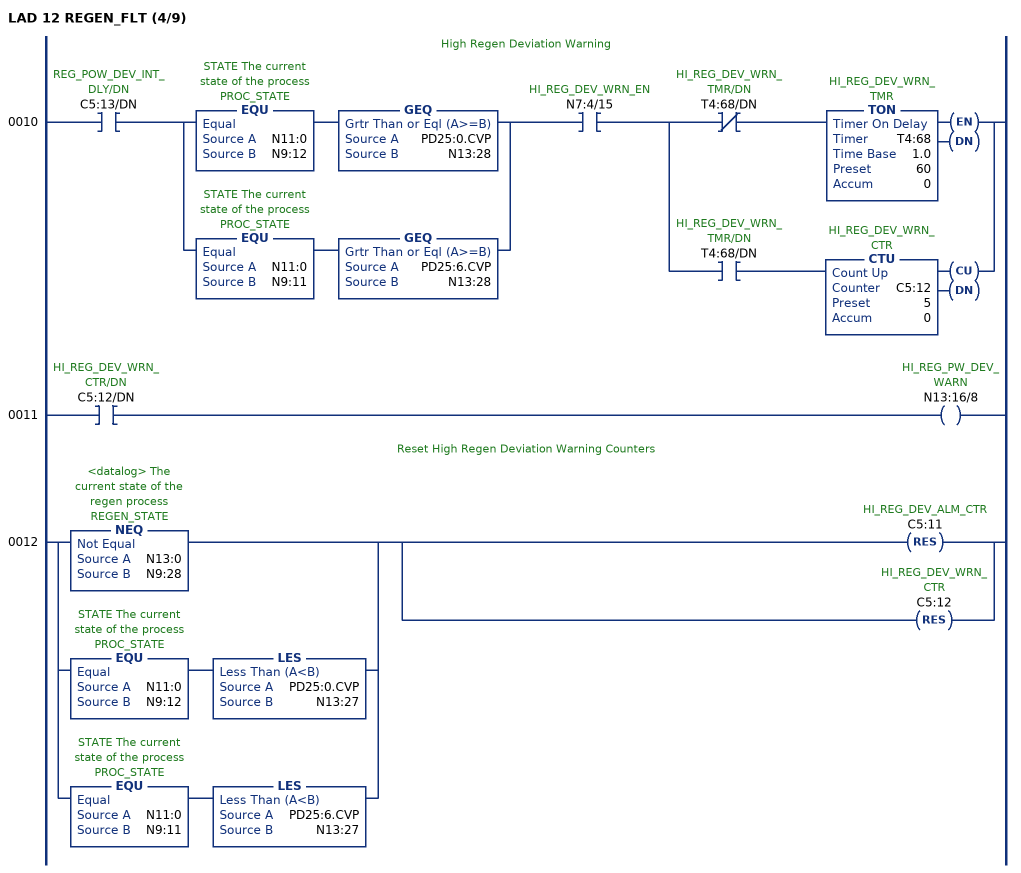
% Rung: 10 %
% High Regen Deviation Warning %
SOR XIC C5:13/DN BST EQU N11:0 N9:12 GEQ PD25:0.CVP N13:28 NXB EQU N11:0 N9:11 GEQ PD25:6.CVP N13:28 BND XIC N7:4/15 BST XIO T4:68/DN TON T4:68 1.0 60 0 NXB XIC T4:68/DN CTU C5:12 5 0 BND EOR
%   C5:13  REG_POW_DEV_INT_DLY %
%   N11:0  PROC_STATE  "STATE The current state of the process" %
%   N9:12  PROC_REGEN_A  "STATE Process Purify B" %
%   N13:28  HI_REG_DEV_WRN_SP %
%   N9:11  PROC_REGEN_B  "STATE Process Purify A" %
%   N7:4/15  HI_REG_DEV_WRN_EN %
%   T4:68  HI_REG_DEV_WRN_TMR %
%   C5:12  HI_REG_DEV_WRN_CTR %
% Rung: 11 %
SOR XIC C5:12/DN OTE N13:16/8 EOR
%   C5:12  HI_REG_DEV_WRN_CTR %
%   N13:16/8  HI_REG_PW_DEV_WARN %
% Rung: 12 %
% Reset High Regen Deviation Warning Counters %
SOR BST NEQ N13:0 N9:28 NXB EQU N11:0 N9:12 LES PD25:0.CVP N13:27 NXB EQU N11:0 N9:11 LES PD25:6.CVP N13:27 BND BST RES C5:11 NXB RES C5:12 BND EOR
%   N13:0  REGEN_STATE  "<datalog> The current state of the regen process" %
%   N9:28  REGEN_RUN %
%   N11:0  PROC_STATE  "STATE The current state of the process" %
%   N9:12  PROC_REGEN_A  "STATE Process Purify B" %
%   N13:27  HI_REG_DEV_ALM_SP %
%   N9:11  PROC_REGEN_B  "STATE Process Purify A" %
%   C5:11  HI_REG_DEV_ALM_CTR %
%   C5:12  HI_REG_DEV_WRN_CTR %

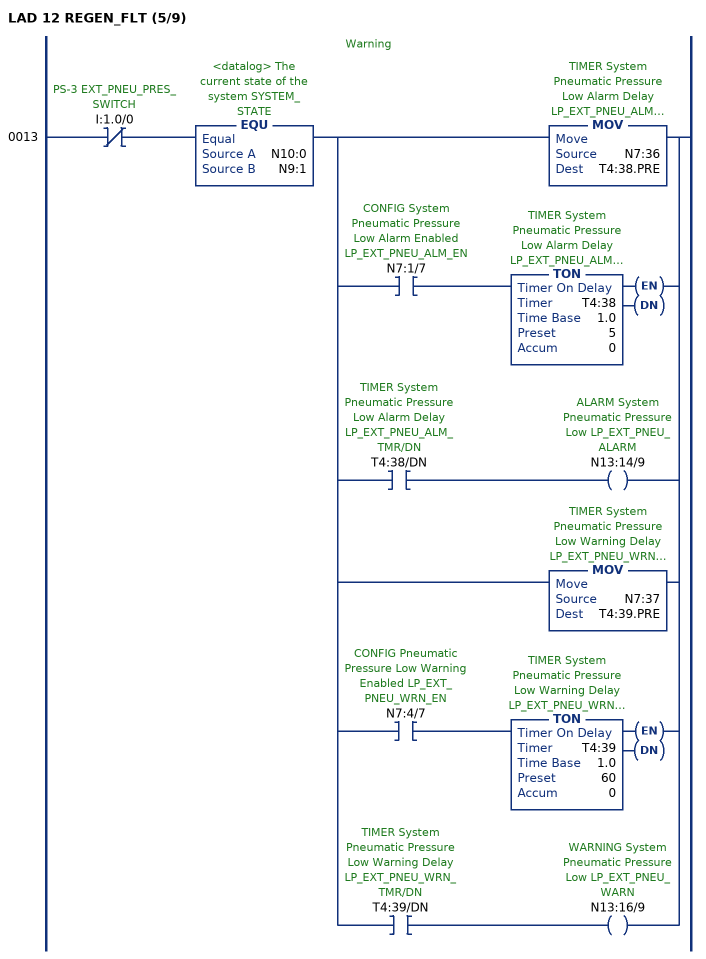
% Rung: 13 %
% Warning %
SOR XIO I:1.0/0 EQU N10:0 N9:1 BST MOV N7:36 T4:38.PRE NXB XIC N7:1/7 TON T4:38 1.0 5 0 NXB XIC T4:38/DN OTE N13:14/9 NXB MOV N7:37 T4:39.PRE NXB XIC N7:4/7 TON T4:39 1.0 60 0 NXB XIC T4:39/DN OTE N13:16/9 BND EOR
%   I:1.0/0  EXT_PNEU_PRES_SWITCH  "PS-3" %
%   N10:0  SYSTEM_STATE  "<datalog> The current state of the system" %
%   N9:1  SYSTEM_PROCESS  "STATE System Process" %
%   N7:36  LP_EXT_PNEU_ALM_DLY  "CONFIG Pneumatic Pressure Low Alarm Delay" %
%   T4:38  LP_EXT_PNEU_ALM_TMR  "TIMER System Pneumatic Pressure Low Alarm Delay" %
%   N7:1/7  LP_EXT_PNEU_ALM_EN  "CONFIG System Pneumatic Pressure Low Alarm Enabled" %
%   N13:14/9  LP_EXT_PNEU_ALARM  "ALARM System Pneumatic Pressure Low" %
%   N7:37  LP_EXT_PNEU_WRN_DLY  "CONFIG Pneumatic Pressure Low Warning Delay" %
%   T4:39  LP_EXT_PNEU_WRN_TMR  "TIMER System Pneumatic Pressure Low Warning Delay" %
%   N7:4/7  LP_EXT_PNEU_WRN_EN  "CONFIG Pneumatic Pressure Low Warning Enabled" %
%   N13:16/9  LP_EXT_PNEU_WARN  "WARNING System Pneumatic Pressure Low" %

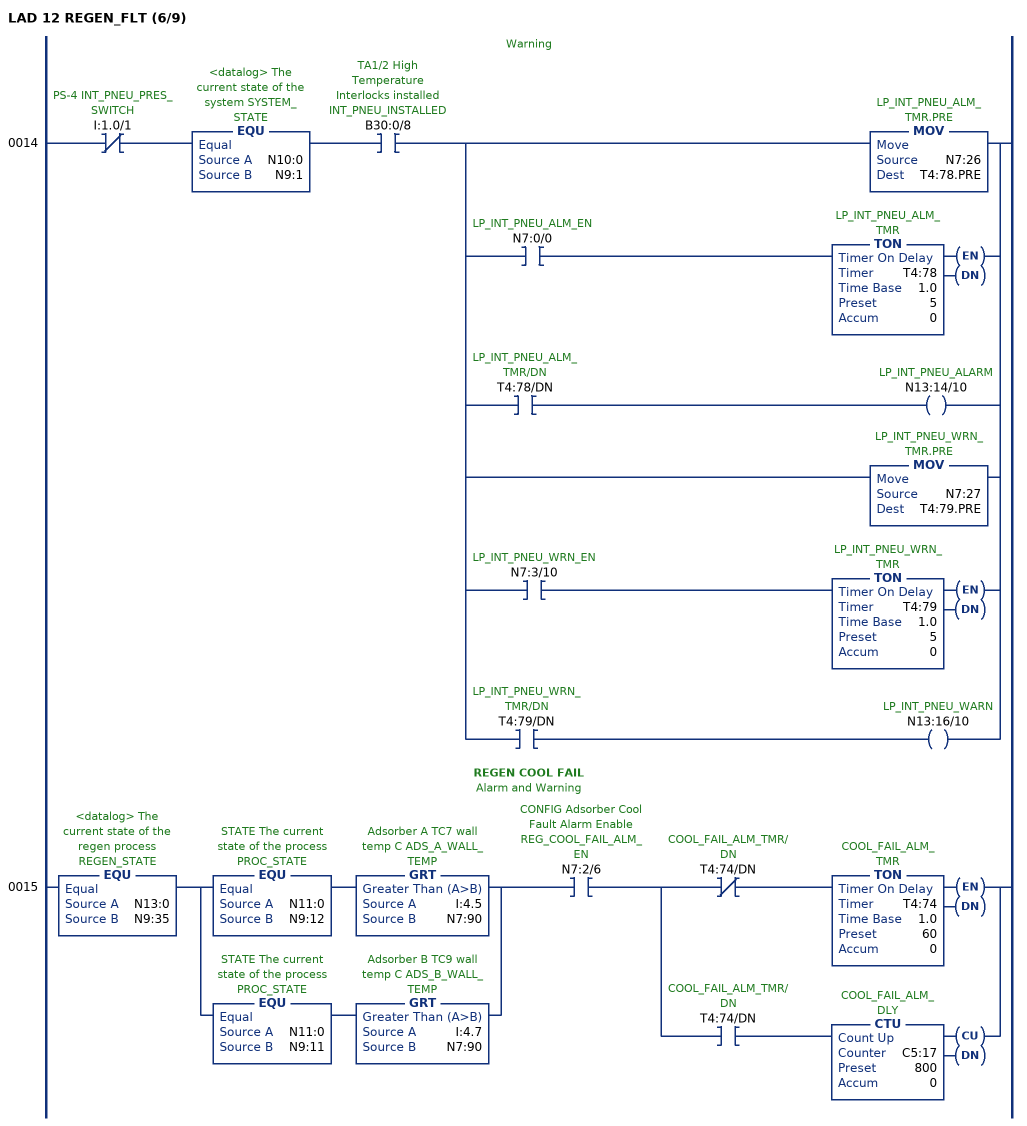
% Rung: 14 %
% Warning %
SOR XIO I:1.0/1 EQU N10:0 N9:1 XIC B30:0/8 BST MOV N7:26 T4:78.PRE NXB XIC N7:0/0 TON T4:78 1.0 5 0 NXB XIC T4:78/DN OTE N13:14/10 NXB MOV N7:27 T4:79.PRE NXB XIC N7:3/10 TON T4:79 1.0 5 0 NXB XIC T4:79/DN OTE N13:16/10 BND EOR
%   I:1.0/1  INT_PNEU_PRES_SWITCH  "PS-4" %
%   N10:0  SYSTEM_STATE  "<datalog> The current state of the system" %
%   N9:1  SYSTEM_PROCESS  "STATE System Process" %
%   B30:0/8  INT_PNEU_INSTALLED  "TA1/2 High Temperature Interlocks installed" %
%   N7:26  LP_INT_PNEU_ALM_DLY %
%   T4:78  LP_INT_PNEU_ALM_TMR %
%   N7:0/0  LP_INT_PNEU_ALM_EN %
%   N13:14/10  LP_INT_PNEU_ALARM %
%   N7:27  LP_INT_PNEU_WRN_DLY %
%   T4:79  LP_INT_PNEU_WRN_TMR %
%   N7:3/10  LP_INT_PNEU_WRN_EN %
%   N13:16/10  LP_INT_PNEU_WARN %
% Rung: 15 %
% TITLE: REGEN COOL FAIL %
% Alarm and Warning %
SOR EQU N13:0 N9:35 BST EQU N11:0 N9:12 GRT I:4.5 N7:90 NXB EQU N11:0 N9:11 GRT I:4.7 N7:90 BND XIC N7:2/6 BST XIO T4:74/DN TON T4:74 1.0 60 0 NXB XIC T4:74/DN CTU C5:17 800 0 BND EOR
%   N13:0  REGEN_STATE  "<datalog> The current state of the regen process" %
%   N9:35  REGEN_COOL_WALL  "STATE Regen Cool wall" %
%   N11:0  PROC_STATE  "STATE The current state of the process" %
%   N9:12  PROC_REGEN_A  "STATE Process Purify B" %
%   I:4.5  ADS_A_WALL_TEMP  "Adsorber A TC7 wall temp C" %
%   N7:90  REG_COOL_FAIL_ALM_SP %
%   N9:11  PROC_REGEN_B  "STATE Process Purify A" %
%   I:4.7  ADS_B_WALL_TEMP  "Adsorber B TC9 wall temp C" %
%   N7:2/6  REG_COOL_FAIL_ALM_EN  "CONFIG Adsorber Cool Fault Alarm Enable" %
%   T4:74  COOL_FAIL_ALM_TMR %
%   C5:17  COOL_FAIL_ALM_DLY %

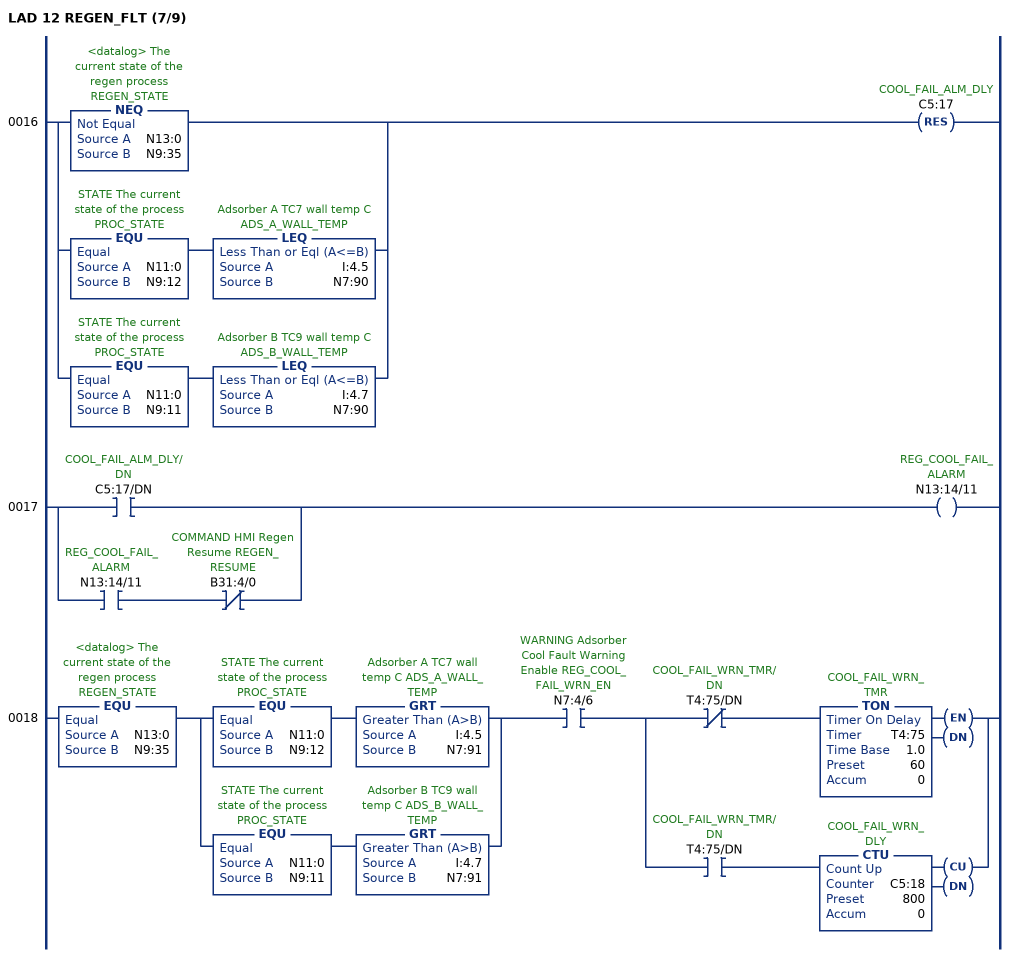
% Rung: 16 %
SOR BST NEQ N13:0 N9:35 NXB EQU N11:0 N9:12 LEQ I:4.5 N7:90 NXB EQU N11:0 N9:11 LEQ I:4.7 N7:90 BND RES C5:17 EOR
%   N13:0  REGEN_STATE  "<datalog> The current state of the regen process" %
%   N9:35  REGEN_COOL_WALL  "STATE Regen Cool wall" %
%   N11:0  PROC_STATE  "STATE The current state of the process" %
%   N9:12  PROC_REGEN_A  "STATE Process Purify B" %
%   I:4.5  ADS_A_WALL_TEMP  "Adsorber A TC7 wall temp C" %
%   N7:90  REG_COOL_FAIL_ALM_SP %
%   N9:11  PROC_REGEN_B  "STATE Process Purify A" %
%   I:4.7  ADS_B_WALL_TEMP  "Adsorber B TC9 wall temp C" %
%   C5:17  COOL_FAIL_ALM_DLY %
% Rung: 17 %
SOR BST XIC C5:17/DN NXB XIC N13:14/11 XIO B31:4/0 BND OTE N13:14/11 EOR
%   C5:17  COOL_FAIL_ALM_DLY %
%   N13:14/11  REG_COOL_FAIL_ALARM %
%   B31:4/0  REGEN_RESUME  "COMMAND HMI Regen Resume" %
% Rung: 18 %
SOR EQU N13:0 N9:35 BST EQU N11:0 N9:12 GRT I:4.5 N7:91 NXB EQU N11:0 N9:11 GRT I:4.7 N7:91 BND XIC N7:4/6 BST XIO T4:75/DN TON T4:75 1.0 60 0 NXB XIC T4:75/DN CTU C5:18 800 0 BND EOR
%   N13:0  REGEN_STATE  "<datalog> The current state of the regen process" %
%   N9:35  REGEN_COOL_WALL  "STATE Regen Cool wall" %
%   N11:0  PROC_STATE  "STATE The current state of the process" %
%   N9:12  PROC_REGEN_A  "STATE Process Purify B" %
%   I:4.5  ADS_A_WALL_TEMP  "Adsorber A TC7 wall temp C" %
%   N7:91  REG_COOL_FAIL_WRN_SP %
%   N9:11  PROC_REGEN_B  "STATE Process Purify A" %
%   I:4.7  ADS_B_WALL_TEMP  "Adsorber B TC9 wall temp C" %
%   N7:4/6  REG_COOL_FAIL_WRN_EN  "WARNING Adsorber Cool Fault Warning Enable" %
%   T4:75  COOL_FAIL_WRN_TMR %
%   C5:18  COOL_FAIL_WRN_DLY %

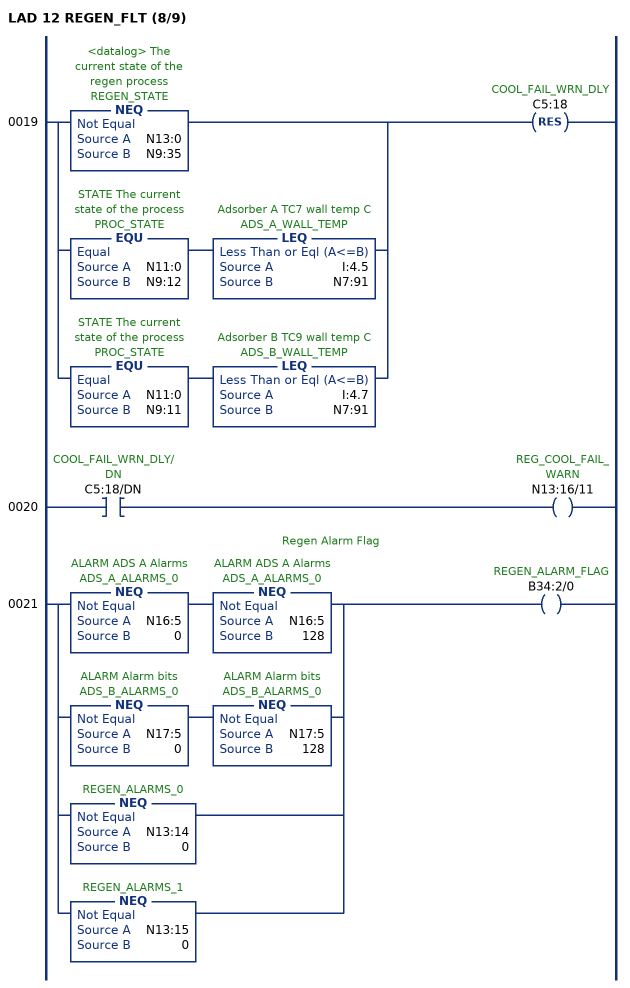
% Rung: 19 %
SOR BST NEQ N13:0 N9:35 NXB EQU N11:0 N9:12 LEQ I:4.5 N7:91 NXB EQU N11:0 N9:11 LEQ I:4.7 N7:91 BND RES C5:18 EOR
%   N13:0  REGEN_STATE  "<datalog> The current state of the regen process" %
%   N9:35  REGEN_COOL_WALL  "STATE Regen Cool wall" %
%   N11:0  PROC_STATE  "STATE The current state of the process" %
%   N9:12  PROC_REGEN_A  "STATE Process Purify B" %
%   I:4.5  ADS_A_WALL_TEMP  "Adsorber A TC7 wall temp C" %
%   N7:91  REG_COOL_FAIL_WRN_SP %
%   N9:11  PROC_REGEN_B  "STATE Process Purify A" %
%   I:4.7  ADS_B_WALL_TEMP  "Adsorber B TC9 wall temp C" %
%   C5:18  COOL_FAIL_WRN_DLY %
% Rung: 20 %
SOR XIC C5:18/DN OTE N13:16/11 EOR
%   C5:18  COOL_FAIL_WRN_DLY %
%   N13:16/11  REG_COOL_FAIL_WARN %
% Rung: 21 %
% Regen Alarm Flag %
SOR BST NEQ N16:5 0 NEQ N16:5 128 NXB NEQ N17:5 0 NEQ N17:5 128 NXB NEQ N13:14 0 NXB NEQ N13:15 0 BND OTE B34:2/0 EOR
%   N16:5  ADS_A_ALARMS_0  "ALARM ADS A Alarms" %
%   N17:5  ADS_B_ALARMS_0  "ALARM Alarm bits" %
%   N13:14  REGEN_ALARMS_0 %
%   N13:15  REGEN_ALARMS_1 %
%   B34:2/0  REGEN_ALARM_FLAG %

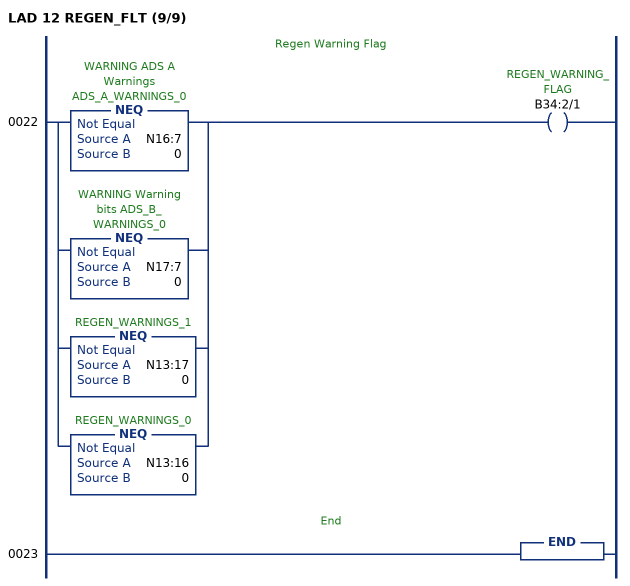
% Rung: 22 %
% Regen Warning Flag %
SOR BST NEQ N16:7 0 NXB NEQ N17:7 0 NXB NEQ N13:17 0 NXB NEQ N13:16 0 BND OTE B34:2/1 EOR
%   N16:7  ADS_A_WARNINGS_0  "WARNING ADS A Warnings" %
%   N17:7  ADS_B_WARNINGS_0  "WARNING Warning bits" %
%   N13:17  REGEN_WARNINGS_1 %
%   N13:16  REGEN_WARNINGS_0 %
%   B34:2/1  REGEN_WARNING_FLAG %
% Rung: 23 %
% End %
SOR END EOR

LADDER 17 "BYPASS"    % Controls the bypass %
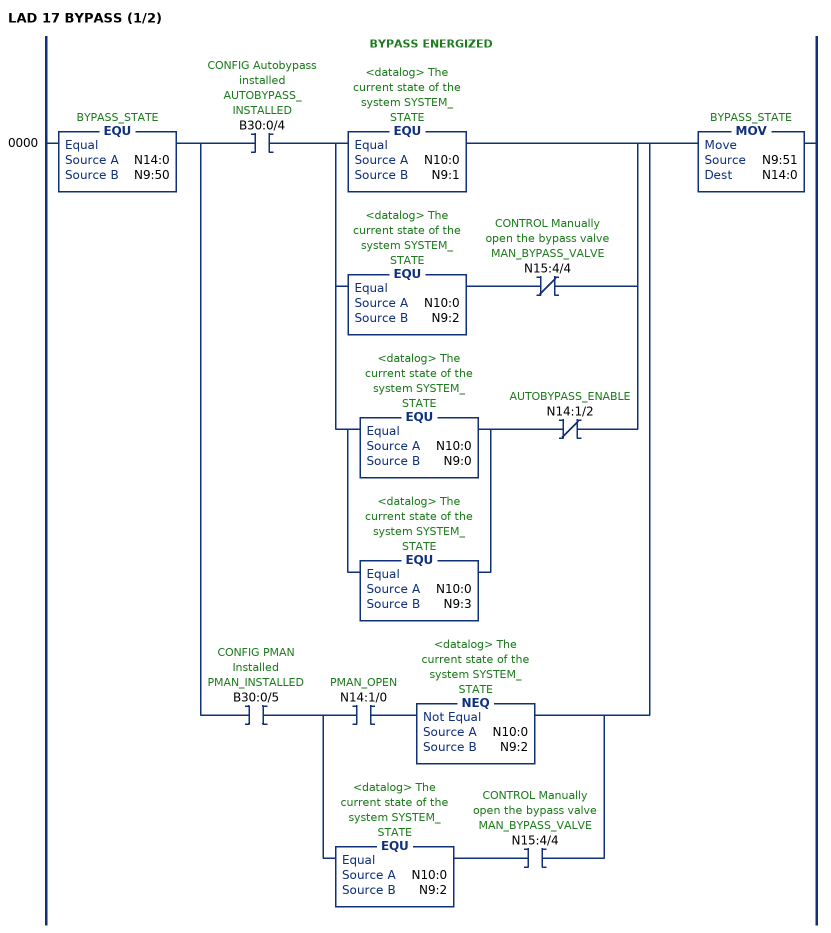
% Rung: 0 %
% TITLE: BYPASS ENERGIZED %
SOR EQU N14:0 N9:50 BST XIC B30:0/4 BST EQU N10:0 N9:1 NXB EQU N10:0 N9:2 XIO N15:4/4 NXB BST EQU N10:0 N9:0 NXB EQU N10:0 N9:3 BND XIO N14:1/2 BND NXB XIC B30:0/5 BST XIC N14:1/0 NEQ N10:0 N9:2 NXB EQU N10:0 N9:2 XIC N15:4/4 BND BND MOV N9:51 N14:0 EOR
%   N14:0  BYPASS_STATE %
%   N9:50  BYPASS_DEENERGIZED  "STATE Bypass Deenergized" %
%   B30:0/4  AUTOBYPASS_INSTALLED  "CONFIG Autobypass installed" %
%   N10:0  SYSTEM_STATE  "<datalog> The current state of the system" %
%   N9:1  SYSTEM_PROCESS  "STATE System Process" %
%   N9:2  SYSTEM_MANUAL  "STATE System Manual" %
%   N15:4/4  MAN_BYPASS_VALVE  "CONTROL Manually open the bypass valve" %
%   N9:0  SYSTEM_STANDBY  "STATE System Standby" %
%   N9:3  SYSTEM_ALARM  "STATE System Alarm" %
%   N14:1/2  AUTOBYPASS_ENABLE %
%   B30:0/5  PMAN_INSTALLED  "CONFIG PMAN Installed" %
%   N14:1/0  PMAN_OPEN %
%   N9:51  BYPASS_ENERGIZED  "STATE Bypass Energized" %

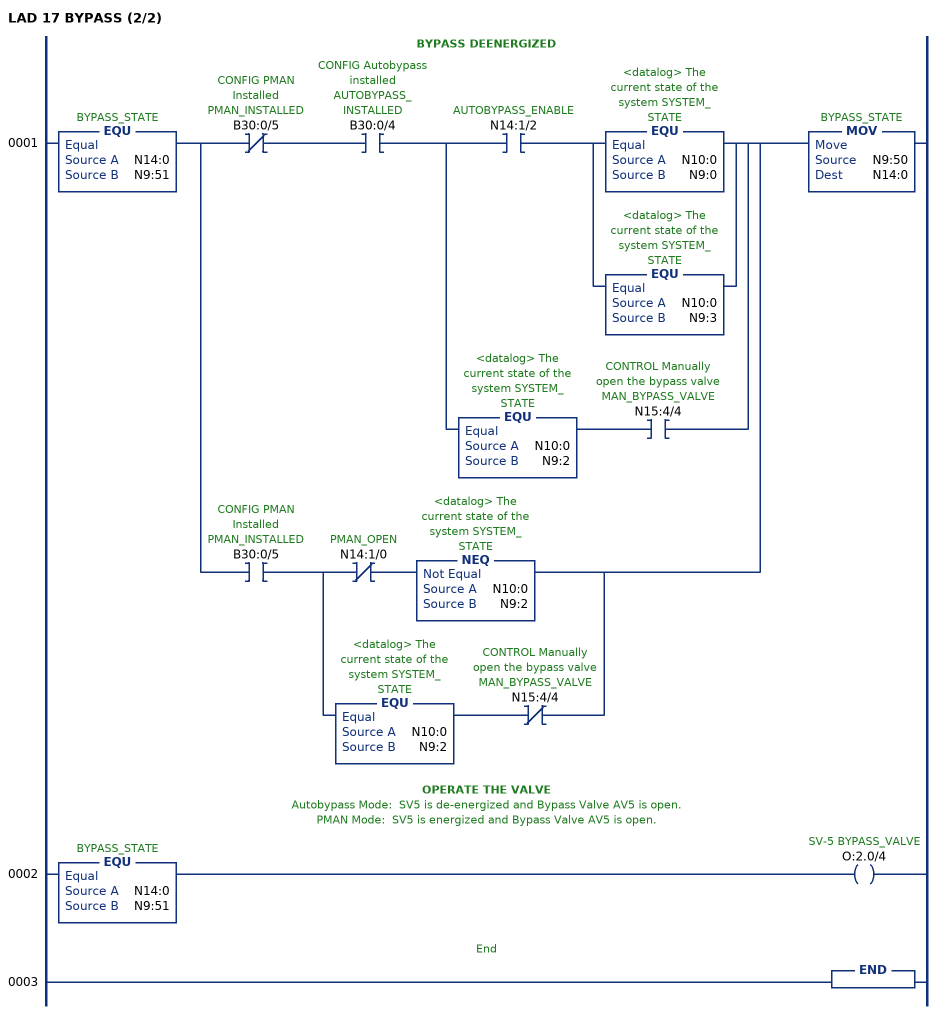
% Rung: 1 %
% TITLE: BYPASS DEENERGIZED %
SOR EQU N14:0 N9:51 BST XIO B30:0/5 XIC B30:0/4 BST XIC N14:1/2 BST EQU N10:0 N9:0 NXB EQU N10:0 N9:3 BND NXB EQU N10:0 N9:2 XIC N15:4/4 BND NXB XIC B30:0/5 BST XIO N14:1/0 NEQ N10:0 N9:2 NXB EQU N10:0 N9:2 XIO N15:4/4 BND BND MOV N9:50 N14:0 EOR
%   N14:0  BYPASS_STATE %
%   N9:51  BYPASS_ENERGIZED  "STATE Bypass Energized" %
%   B30:0/5  PMAN_INSTALLED  "CONFIG PMAN Installed" %
%   B30:0/4  AUTOBYPASS_INSTALLED  "CONFIG Autobypass installed" %
%   N14:1/2  AUTOBYPASS_ENABLE %
%   N10:0  SYSTEM_STATE  "<datalog> The current state of the system" %
%   N9:0  SYSTEM_STANDBY  "STATE System Standby" %
%   N9:3  SYSTEM_ALARM  "STATE System Alarm" %
%   N9:2  SYSTEM_MANUAL  "STATE System Manual" %
%   N15:4/4  MAN_BYPASS_VALVE  "CONTROL Manually open the bypass valve" %
%   N14:1/0  PMAN_OPEN %
%   N9:50  BYPASS_DEENERGIZED  "STATE Bypass Deenergized" %
% Rung: 2 %
% TITLE: OPERATE THE VALVE %
% Autobypass Mode:  SV5 is de-energized and Bypass Valve AV5 is open.
% PMAN Mode:  SV5 is energized and Bypass Valve AV5 is open. %
SOR EQU N14:0 N9:51 OTE O:2.0/4 EOR
%   N14:0  BYPASS_STATE %
%   N9:51  BYPASS_ENERGIZED  "STATE Bypass Energized" %
%   O:2.0/4  BYPASS_VALVE  "SV-5" %
% Rung: 3 %
% End %
SOR END EOR

LADDER 20 "ADS_A"    % Controls the Adsorber A %
